LIN {X 0,Y 676.255,Z 793.272,A -85,B 0,C 180,E1 -4017.987,E2 -4017.987} C_VEL
LIN {X 0,Y 675.529,Z 814.442,A -85,B 0,C 180,E1 -4018.503,E2 -4018.503} C_VEL
LIN {X 0,Y 674.622,Z 838.545,A -85,B 0,C 180,E1 -4019.247,E2 -4019.247} C_VEL
LIN {X 0,Y 673.655,Z 859.341,A -85,B 0,C 180,E1 -4020.036,E2 -4020.036} C_VEL
LIN {X 0,Y 672.656,Z 880.169,A -85,B 0,C 180,E1 -4020.961,E2 -4020.961} C_VEL
LIN {X 0,Y 671.429,Z 902.312,A -85,B 0,C 180,E1 -4022.121,E2 -4022.121} C_VEL
LIN {X 0,Y 670.354,Z 922.188,A -85,B 0,C 180,E1 -4023.323,E2 -4023.323} C_VEL
LIN {X 0,Y 669.168,Z 942.613,A -85,B 0,C 180,E1 -4024.748,E2 -4024.748} C_VEL
LIN {X 0,Y 668.228,Z 959.686,A -85,B 0,C 180,E1 -4026.101,E2 -4026.101} C_VEL
LIN {X 0,Y 667.192,Z 978.605,A -85,B 0,C 180,E1 -4027.811,E2 -4027.811} C_VEL
LIN {X 0,Y 666.434,Z 993.632,A -85,B 0,C 180,E1 -4029.354,E2 -4029.354} C_VEL
LIN {X 0,Y 665.654,Z 1009.818,A -85,B 0,C 180,E1 -4031.249,E2 -4031.249} C_VEL
LIN {X 0,Y 665.144,Z 1022.543,A -85,B 0,C 180,E1 -4032.957,E2 -4032.957} C_VEL
LIN {X 0,Y 664.665,Z 1035.765,A -85,B 0,C 180,E1 -4035.004,E2 -4035.004} C_VEL
LIN {X 0,Y 664.369,Z 1045.92,A -85,B 0,C 180,E1 -4036.844,E2 -4036.844} C_VEL
LIN {X 0,Y 664.132,Z 1055.929,A -85,B 0,C 180,E1 -4039.001,E2 -4039.001} C_VEL
LIN {X 0,Y 664.022,Z 1062.817,A -85,B 0,C 180,E1 -4040.815,E2 -4040.815} C_VEL
LIN {X 0,Y 663.962,Z 1069.244,A -85,B 0,C 180,E1 -4042.907,E2 -4042.907} C_VEL
LIN {X 0,Y 663.925,Z 1073.656,A -85,B 0,C 180,E1 -4044.902,E2 -4044.902} C_VEL
LIN {X 0,Y 663.917,Z 1076.574,A -85,B 0,C 180,E1 -4046.806,E2 -4046.806} C_VEL
LIN {X 0,Y 663.91,Z 1078.26,A -85,B 0,C 180,E1 -4049.051,E2 -4049.051} C_VEL
LIN {X 0,Y 663.905,Z 1078.283,A -85,B 0,C 180,E1 -4050.863,E2 -4050.863} C_VEL
LIN {X 0,Y 663.916,Z 1076.799,A -85,B 0,C 180,E1 -4053.021,E2 -4053.021} C_VEL
LIN {X 0,Y 663.925,Z 1073.815,A -85,B 0,C 180,E1 -4055.011,E2 -4055.011} C_VEL
LIN {X 0,Y 663.956,Z 1069.451,A -85,B 0,C 180,E1 -4057.006,E2 -4057.006} C_VEL
LIN {X 0,Y 664.011,Z 1063.12,A -85,B 0,C 180,E1 -4059.097,E2 -4059.097} C_VEL
LIN {X 0,Y 664.128,Z 1056.187,A -85,B 0,C 180,E1 -4060.935,E2 -4060.935} C_VEL
LIN {X 0,Y 664.355,Z 1046.484,A -85,B 0,C 180,E1 -4063.047,E2 -4063.047} C_VEL
LIN {X 0,Y 664.649,Z 1036.288,A -85,B 0,C 180,E1 -4064.907,E2 -4064.907} C_VEL
LIN {X 0,Y 665.121,Z 1023.161,A -85,B 0,C 180,E1 -4066.956,E2 -4066.956} C_VEL
LIN {X 0,Y 665.624,Z 1010.525,A -85,B 0,C 180,E1 -4068.661,E2 -4068.661} C_VEL
LIN {X 0,Y 666.403,Z 994.378,A -85,B 0,C 180,E1 -4070.565,E2 -4070.565} C_VEL
LIN {X 0,Y 667.168,Z 979.013,A -85,B 0,C 180,E1 -4072.149,E2 -4072.149} C_VEL
LIN {X 0,Y 668.189,Z 960.507,A -85,B 0,C 180,E1 -4073.83,E2 -4073.83} C_VEL
LIN {X 0,Y 669.128,Z 943.221,A -85,B 0,C 180,E1 -4075.206,E2 -4075.206} C_VEL
LIN {X 0,Y 670.317,Z 922.91,A -85,B 0,C 180,E1 -4076.631,E2 -4076.631} C_VEL
LIN {X 0,Y 671.389,Z 903.049,A -85,B 0,C 180,E1 -4077.837,E2 -4077.837} C_VEL
LIN {X 0,Y 672.604,Z 881.269,A -85,B 0,C 180,E1 -4078.988,E2 -4078.988} C_VEL
LIN {X 0,Y 673.605,Z 860.478,A -85,B 0,C 180,E1 -4079.917,E2 -4079.917} C_VEL
LIN {X 0,Y 674.538,Z 840.352,A -85,B 0,C 180,E1 -4080.688,E2 -4080.688} C_VEL
LIN {X 0,Y 675.503,Z 815.102,A -85,B 0,C 180,E1 -4081.479,E2 -4081.479} C_VEL
LIN {X 0,Y 676.234,Z 793.804,A -85,B 0,C 180,E1 -4082.002,E2 -4082.002} C_VEL
LIN {X 0,Y 676.909,Z 768.362,A -85,B 0,C 180,E1 -4082.466,E2 -4082.466} C_VEL
LIN {X 0,Y 677.775,Z 687.285,A -85,B 0,C 180,E1 -4083.452,E2 -4083.452} C_VEL
LIN {X 0,Y 680.315,Z 434.11,A -85,B 0,C 180,E1 -4086.498,E2 -4086.498} C_VEL
LIN {X 0,Y 680.519,Z 397.747,A -85,B 0,C 180,E1 -4086.954,E2 -4086.954} C_VEL
LIN {X 0,Y 675.309,Z 375.993,A -85,B 0,C 180,E1 -4087.591,E2 -4087.591} C_VEL
LIN {X 0,Y 675.512,Z 367.277,A -85,B 0,C 180,E1 -4088.256,E2 -4088.256} C_VEL
LIN {X 0,Y 667.876,Z 347.353,A -85,B 0,C 180,E1 -4090.356,E2 -4090.356} C_VEL
LIN {X 0,Y 664.606,Z 338.448,A -85,B 0,C 180,E1 -4091.345,E2 -4091.345} C_VEL
LIN {X 0,Y 664.58,Z 338.444,A -85,B 0,C 180,E1 -4094.035,E2 -4094.035} C_VEL
LIN {X 0,Y 664.647,Z 338.444,A -85,B 0,C 180,E1 -4097.04,E2 -4097.04} C_VEL
LIN {X 0,Y 664.579,Z 338.44,A -85,B 0,C 180,E1 -4099.913,E2 -4099.913} C_VEL
LIN {X 0,Y 664.625,Z 338.437,A -85,B 0,C 180,E1 -4102.735,E2 -4102.735} C_VEL
LIN {X 0,Y 664.588,Z 338.439,A -85,B 0,C 180,E1 -4105.842,E2 -4105.842} C_VEL
LIN {X 0,Y 664.593,Z 338.436,A -85,B 0,C 180,E1 -4108.546,E2 -4108.546} C_VEL
LIN {X 0,Y 664.605,Z 338.436,A -85,B 0,C 180,E1 -4111.711,E2 -4111.711} C_VEL
LIN {X 0,Y 664.584,Z 338.441,A -85,B 0,C 180,E1 -4114.418,E2 -4114.418} C_VEL
LIN {X 0,Y 664.651,Z 338.44,A -85,B 0,C 180,E1 -4117.472,E2 -4117.472} C_VEL
LIN {X 0,Y 664.579,Z 338.438,A -85,B 0,C 180,E1 -4120.396,E2 -4120.396} C_VEL
LIN {X 0,Y 664.647,Z 338.438,A -85,B 0,C 180,E1 -4123.301,E2 -4123.301} C_VEL
LIN {X 0,Y 664.586,Z 338.442,A -85,B 0,C 180,E1 -4126.248,E2 -4126.248} C_VEL
LIN {X 0,Y 664.604,Z 338.433,A -85,B 0,C 180,E1 -4128.985,E2 -4128.985} C_VEL
LIN {X 0,Y 664.6,Z 338.434,A -85,B 0,C 180,E1 -4132.131,E2 -4132.131} C_VEL
LIN {X 0,Y 664.589,Z 338.44,A -85,B 0,C 180,E1 -4134.869,E2 -4134.869} C_VEL
LIN {X 0,Y 664.636,Z 338.436,A -85,B 0,C 180,E1 -4137.931,E2 -4137.931} C_VEL
LIN {X 0,Y 664.582,Z 338.439,A -85,B 0,C 180,E1 -4140.776,E2 -4140.776} C_VEL
LIN {X 0,Y 664.649,Z 338.435,A -85,B 0,C 180,E1 -4143.709,E2 -4143.709} C_VEL
LIN {X 0,Y 664.584,Z 338.434,A -85,B 0,C 180,E1 -4146.653,E2 -4146.653} C_VEL
LIN {X 0,Y 664.618,Z 338.439,A -85,B 0,C 180,E1 -4149.438,E2 -4149.438} C_VEL
LIN {X 0,Y 664.594,Z 338.443,A -85,B 0,C 180,E1 -4152.601,E2 -4152.601} C_VEL
LIN {X 0,Y 664.598,Z 338.435,A -85,B 0,C 180,E1 -4155.355,E2 -4155.355} C_VEL
LIN {X 0,Y 664.611,Z 338.441,A -85,B 0,C 180,E1 -4158.509,E2 -4158.509} C_VEL
LIN {X 0,Y 664.589,Z 338.439,A -85,B 0,C 180,E1 -4161.259,E2 -4161.259} C_VEL
LIN {X 0,Y 664.647,Z 338.435,A -85,B 0,C 180,E1 -4164.264,E2 -4164.264} C_VEL
LIN {X 0,Y 664.585,Z 338.438,A -85,B 0,C 180,E1 -4167.121,E2 -4167.121} C_VEL
LIN {X 0,Y 664.643,Z 338.438,A -85,B 0,C 180,E1 -4169.965,E2 -4169.965} C_VEL
LIN {X 0,Y 664.591,Z 338.442,A -85,B 0,C 180,E1 -4173.069,E2 -4173.069} C_VEL
LIN {X 0,Y 664.624,Z 338.437,A -85,B 0,C 180,E1 -4175.926,E2 -4175.926} C_VEL
LIN {X 0,Y 664.65,Z 338.441,A -85,B 0,C 180,E1 -4176.376,E2 -4176.376} C_VEL
LIN {X 0,Y 663.65,Z 338.574,A -85,B 0,C 180,E1 -4177.041,E2 -4177.041} C_VEL
LIN {X 0,Y 657.182,Z 339.37,A -85,B 0,C 180,E1 -4178.902,E2 -4178.902} C_VEL
LIN {X 0,Y 656.649,Z 339.431,A -85,B 0,C 180,E1 -4179.386,E2 -4179.386} C_VEL
LIN {X 0,Y 656.711,Z 339.43,A -85,B 0,C 180,E1 -4182.298,E2 -4182.298} C_VEL
LIN {X 0,Y 656.652,Z 339.432,A -85,B 0,C 180,E1 -4185.325,E2 -4185.325} C_VEL
LIN {X 0,Y 656.7,Z 339.431,A -85,B 0,C 180,E1 -4188.252,E2 -4188.252} C_VEL
LIN {X 0,Y 656.721,Z 339.5,A -85,B 0,C 180,E1 -4190.391,E2 -4190.391} C_VEL
LIN {X 0,Y 660.252,Z 349.072,A -85,B 0,C 180,E1 -4191.479,E2 -4191.479} C_VEL
LIN {X 0,Y 674.214,Z 372.691,A -85,B 0,C 180,E1 -4192.737,E2 -4192.737} C_VEL
LIN {X 0,Y 672.117,Z 564.734,A -85,B 0,C 180,E1 -4195.097,E2 -4195.097} C_VEL
LIN {X 0,Y 670.164,Z 737.365,A -85,B 0,C 180,E1 -4197.196,E2 -4197.196} C_VEL
LIN {X 0,Y 669.465,Z 762.862,A -85,B 0,C 180,E1 -4197.658,E2 -4197.658} C_VEL
LIN {X 0,Y 668.692,Z 783.876,A -85,B 0,C 180,E1 -4198.172,E2 -4198.172} C_VEL
LIN {X 0,Y 667.724,Z 807.392,A -85,B 0,C 180,E1 -4198.894,E2 -4198.894} C_VEL
LIN {X 0,Y 666.664,Z 828.321,A -85,B 0,C 180,E1 -4199.689,E2 -4199.689} C_VEL
LIN {X 0,Y 665.591,Z 849.051,A -85,B 0,C 180,E1 -4200.612,E2 -4200.612} C_VEL
LIN {X 0,Y 664.244,Z 871.561,A -85,B 0,C 180,E1 -4201.793,E2 -4201.793} C_VEL
LIN {X 0,Y 663.077,Z 891.047,A -85,B 0,C 180,E1 -4202.976,E2 -4202.976} C_VEL
LIN {X 0,Y 661.793,Z 911.734,A -85,B 0,C 180,E1 -4204.422,E2 -4204.422} C_VEL
LIN {X 0,Y 660.725,Z 928.876,A -85,B 0,C 180,E1 -4205.788,E2 -4205.788} C_VEL
LIN {X 0,Y 659.58,Z 948.163,A -85,B 0,C 180,E1 -4207.541,E2 -4207.541} C_VEL
LIN {X 0,Y 658.72,Z 963.223,A -85,B 0,C 180,E1 -4209.102,E2 -4209.102} C_VEL
LIN {X 0,Y 657.874,Z 979.475,A -85,B 0,C 180,E1 -4211.019,E2 -4211.019} C_VEL
LIN {X 0,Y 657.298,Z 992.211,A -85,B 0,C 180,E1 -4212.744,E2 -4212.744} C_VEL
LIN {X 0,Y 656.756,Z 1005.695,A -85,B 0,C 180,E1 -4214.851,E2 -4214.851} C_VEL
LIN {X 0,Y 656.432,Z 1015.336,A -85,B 0,C 180,E1 -4216.613,E2 -4216.613} C_VEL
LIN {X 0,Y 656.186,Z 1024.942,A -85,B 0,C 180,E1 -4218.664,E2 -4218.664} C_VEL
LIN {X 0,Y 656.047,Z 1032.359,A -85,B 0,C 180,E1 -4220.614,E2 -4220.614} C_VEL
LIN {X 0,Y 655.948,Z 1038.123,A -85,B 0,C 180,E1 -4222.467,E2 -4222.467} C_VEL
LIN {X 0,Y 655.915,Z 1043.254,A -85,B 0,C 180,E1 -4224.664,E2 -4224.664} C_VEL
LIN {X 0,Y 655.912,Z 1046.179,A -85,B 0,C 180,E1 -4226.504,E2 -4226.504} C_VEL
LIN {X 0,Y 655.898,Z 1048.129,A -85,B 0,C 180,E1 -4228.602,E2 -4228.602} C_VEL
LIN {X 0,Y 655.894,Z 1048.362,A -85,B 0,C 180,E1 -4230.612,E2 -4230.612} C_VEL
LIN {X 0,Y 655.907,Z 1047.397,A -85,B 0,C 180,E1 -4232.446,E2 -4232.446} C_VEL
LIN {X 0,Y 655.918,Z 1044.691,A -85,B 0,C 180,E1 -4234.634,E2 -4234.634} C_VEL
LIN {X 0,Y 655.93,Z 1040.795,A -85,B 0,C 180,E1 -4236.565,E2 -4236.565} C_VEL
LIN {X 0,Y 655.988,Z 1035.585,A -85,B 0,C 180,E1 -4238.503,E2 -4238.503} C_VEL
LIN {X 0,Y 656.123,Z 1028.137,A -85,B 0,C 180,E1 -4240.626,E2 -4240.626} C_VEL
LIN {X 0,Y 656.298,Z 1020.469,A -85,B 0,C 180,E1 -4242.422,E2 -4242.422} C_VEL
LIN {X 0,Y 656.627,Z 1009.634,A -85,B 0,C 180,E1 -4244.552,E2 -4244.552} C_VEL
LIN {X 0,Y 657.016,Z 998.83,A -85,B 0,C 180,E1 -4246.353,E2 -4246.353} C_VEL
LIN {X 0,Y 657.631,Z 985.069,A -85,B 0,C 180,E1 -4248.345,E2 -4248.345} C_VEL
LIN {X 0,Y 658.286,Z 971.227,A -85,B 0,C 180,E1 -4250.077,E2 -4250.077} C_VEL
LIN {X 0,Y 659.186,Z 955.439,A -85,B 0,C 180,E1 -4251.825,E2 -4251.825} C_VEL
LIN {X 0,Y 660.116,Z 938.8,A -85,B 0,C 180,E1 -4253.429,E2 -4253.429} C_VEL
LIN {X 0,Y 661.281,Z 920.46,A -85,B 0,C 180,E1 -4255,E2 -4255} C_VEL
LIN {X 0,Y 662.437,Z 901.028,A -85,B 0,C 180,E1 -4256.441,E2 -4256.441} C_VEL
LIN {X 0,Y 663.767,Z 880.336,A -85,B 0,C 180,E1 -4257.79,E2 -4257.79} C_VEL
LIN {X 0,Y 664.964,Z 859.37,A -85,B 0,C 180,E1 -4258.959,E2 -4258.959} C_VEL
LIN {X 0,Y 666.25,Z 837.109,A -85,B 0,C 180,E1 -4260.034,E2 -4260.034} C_VEL
LIN {X 0,Y 667.326,Z 815.541,A -85,B 0,C 180,E1 -4260.899,E2 -4260.899} C_VEL
LIN {X 0,Y 668.244,Z 795.426,A -85,B 0,C 180,E1 -4261.581,E2 -4261.581} C_VEL
LIN {X 0,Y 669.182,Z 770.572,A -85,B 0,C 180,E1 -4262.26,E2 -4262.26} C_VEL
LIN {X 0,Y 669.871,Z 748.473,A -85,B 0,C 180,E1 -4262.713,E2 -4262.713} C_VEL
LIN {X 0,Y 670.423,Z 721.817,A -85,B 0,C 180,E1 -4263.101,E2 -4263.101} C_VEL
LIN {X 0,Y 673.237,Z 466.687,A -85,B 0,C 180,E1 -4266.188,E2 -4266.188} C_VEL
LIN {X 0,Y 674.129,Z 372.539,A -85,B 0,C 180,E1 -4267.361,E2 -4267.361} C_VEL
LIN {X 0,Y 662.253,Z 352.49,A -85,B 0,C 180,E1 -4268.425,E2 -4268.425} C_VEL
LIN {X 0,Y 659.963,Z 348.582,A -85,B 0,C 180,E1 -4268.646,E2 -4268.646} C_VEL
LIN {X 0,Y 656.696,Z 339.429,A -85,B 0,C 180,E1 -4269.743,E2 -4269.743} C_VEL
LIN {X 0,Y 656.642,Z 339.436,A -85,B 0,C 180,E1 -4272.539,E2 -4272.539} C_VEL
LIN {X 0,Y 656.706,Z 339.422,A -85,B 0,C 180,E1 -4275.444,E2 -4275.444} C_VEL
LIN {X 0,Y 656.644,Z 339.408,A -85,B 0,C 180,E1 -4278.401,E2 -4278.401} C_VEL
LIN {X 0,Y 656.666,Z 339.432,A -85,B 0,C 180,E1 -4281.145,E2 -4281.145} C_VEL
LIN {X 0,Y 656.657,Z 339.431,A -85,B 0,C 180,E1 -4284.324,E2 -4284.324} C_VEL
LIN {X 0,Y 656.651,Z 339.432,A -85,B 0,C 180,E1 -4287.07,E2 -4287.07} C_VEL
LIN {X 0,Y 656.679,Z 339.429,A -85,B 0,C 180,E1 -4290.217,E2 -4290.217} C_VEL
LIN {X 0,Y 656.643,Z 339.424,A -85,B 0,C 180,E1 -4293.014,E2 -4293.014} C_VEL
LIN {X 0,Y 656.709,Z 339.42,A -85,B 0,C 180,E1 -4296.013,E2 -4296.013} C_VEL
LIN {X 0,Y 656.639,Z 339.431,A -85,B 0,C 180,E1 -4298.939,E2 -4298.939} C_VEL
LIN {X 0,Y 656.702,Z 339.43,A -85,B 0,C 180,E1 -4301.823,E2 -4301.823} C_VEL
LIN {X 0,Y 656.643,Z 339.422,A -85,B 0,C 180,E1 -4304.887,E2 -4304.887} C_VEL
LIN {X 0,Y 656.665,Z 339.434,A -85,B 0,C 180,E1 -4307.602,E2 -4307.602} C_VEL
LIN {X 0,Y 656.654,Z 339.429,A -85,B 0,C 180,E1 -4310.8,E2 -4310.8} C_VEL
LIN {X 0,Y 656.649,Z 339.427,A -85,B 0,C 180,E1 -4313.53,E2 -4313.53} C_VEL
LIN {X 0,Y 656.675,Z 339.426,A -85,B 0,C 180,E1 -4316.683,E2 -4316.683} C_VEL
LIN {X 0,Y 656.641,Z 339.426,A -85,B 0,C 180,E1 -4319.477,E2 -4319.477} C_VEL
LIN {X 0,Y 656.708,Z 339.418,A -85,B 0,C 180,E1 -4322.443,E2 -4322.443} C_VEL
LIN {X 0,Y 656.639,Z 339.431,A -85,B 0,C 180,E1 -4325.417,E2 -4325.417} C_VEL
LIN {X 0,Y 656.709,Z 339.422,A -85,B 0,C 180,E1 -4328.317,E2 -4328.317} C_VEL
LIN {X 0,Y 656.642,Z 339.427,A -85,B 0,C 180,E1 -4331.328,E2 -4331.328} C_VEL
LIN {X 0,Y 656.67,Z 339.431,A -85,B 0,C 180,E1 -4334.101,E2 -4334.101} C_VEL
LIN {X 0,Y 656.65,Z 339.425,A -85,B 0,C 180,E1 -4337.273,E2 -4337.273} C_VEL
LIN {X 0,Y 656.648,Z 339.431,A -85,B 0,C 180,E1 -4339.943,E2 -4339.943} C_VEL
LIN {X 0,Y 656.685,Z 339.426,A -85,B 0,C 180,E1 -4343.037,E2 -4343.037} C_VEL
LIN {X 0,Y 656.64,Z 339.43,A -85,B 0,C 180,E1 -4345.85,E2 -4345.85} C_VEL
LIN {X 0,Y 656.717,Z 339.428,A -85,B 0,C 180,E1 -4348.859,E2 -4348.859} C_VEL
LIN {X 0,Y 656.638,Z 339.428,A -85,B 0,C 180,E1 -4351.794,E2 -4351.794} C_VEL
LIN {X 0,Y 656.689,Z 339.428,A -85,B 0,C 180,E1 -4354.607,E2 -4354.607} C_VEL
LIN {X 0,Y 656.649,Z 339.431,A -85,B 0,C 180,E1 -4357.645,E2 -4357.645} C_VEL
LIN {X 0,Y 656.648,Z 339.416,A -85,B 0,C 180,E1 -4360.328,E2 -4360.328} C_VEL
LIN {X 0,Y 656.671,Z 339.428,A -85,B 0,C 180,E1 -4363.492,E2 -4363.492} C_VEL
LIN {X 0,Y 656.642,Z 339.431,A -85,B 0,C 180,E1 -4366.265,E2 -4366.265} C_VEL
LIN {X 0,Y 656.658,Z 339.573,A -85,B 0,C 180,E1 -4368.184,E2 -4368.184} C_VEL
LIN {X 0,Y 666.139,Z 364.38,A -85,B 0,C 180,E1 -4370.899,E2 -4370.899} C_VEL
LIN {X 0,Y 668.561,Z 371.173,A -85,B 0,C 180,E1 -4371.6,E2 -4371.6} C_VEL
LIN {X 0,Y 668.498,Z 376.61,A -85,B 0,C 180,E1 -4371.992,E2 -4371.992} C_VEL
LIN {X 0,Y 674.27,Z 401.056,A -85,B 0,C 180,E1 -4372.692,E2 -4372.692} C_VEL
LIN {X 0,Y 671.314,Z 665.846,A -85,B 0,C 180,E1 -4375.914,E2 -4375.914} C_VEL
LIN {X 0,Y 670.159,Z 767.706,A -85,B 0,C 180,E1 -4377.156,E2 -4377.156} C_VEL
LIN {X 0,Y 669.461,Z 793.009,A -85,B 0,C 180,E1 -4377.616,E2 -4377.616} C_VEL
LIN {X 0,Y 668.687,Z 814.006,A -85,B 0,C 180,E1 -4378.131,E2 -4378.131} C_VEL
LIN {X 0,Y 667.733,Z 837.257,A -85,B 0,C 180,E1 -4378.844,E2 -4378.844} C_VEL
LIN {X 0,Y 666.671,Z 858.206,A -85,B 0,C 180,E1 -4379.639,E2 -4379.639} C_VEL
LIN {X 0,Y 665.63,Z 878.269,A -85,B 0,C 180,E1 -4380.53,E2 -4380.53} C_VEL
LIN {X 0,Y 664.255,Z 901.416,A -85,B 0,C 180,E1 -4381.739,E2 -4381.739} C_VEL
LIN {X 0,Y 663.095,Z 920.727,A -85,B 0,C 180,E1 -4382.91,E2 -4382.91} C_VEL
LIN {X 0,Y 661.775,Z 942.002,A -85,B 0,C 180,E1 -4384.398,E2 -4384.398} C_VEL
LIN {X 0,Y 660.695,Z 959.399,A -85,B 0,C 180,E1 -4385.787,E2 -4385.787} C_VEL
LIN {X 0,Y 659.552,Z 978.604,A -85,B 0,C 180,E1 -4387.54,E2 -4387.54} C_VEL
LIN {X 0,Y 658.705,Z 993.63,A -85,B 0,C 180,E1 -4389.101,E2 -4389.101} C_VEL
LIN {X 0,Y 657.857,Z 1009.82,A -85,B 0,C 180,E1 -4391.018,E2 -4391.018} C_VEL
LIN {X 0,Y 657.284,Z 1022.521,A -85,B 0,C 180,E1 -4392.744,E2 -4392.744} C_VEL
LIN {X 0,Y 656.744,Z 1035.973,A -85,B 0,C 180,E1 -4394.855,E2 -4394.855} C_VEL
LIN {X 0,Y 656.42,Z 1046.022,A -85,B 0,C 180,E1 -4396.702,E2 -4396.702} C_VEL
LIN {X 0,Y 656.155,Z 1056.164,A -85,B 0,C 180,E1 -4398.924,E2 -4398.924} C_VEL
LIN {X 0,Y 656.032,Z 1063.12,A -85,B 0,C 180,E1 -4400.791,E2 -4400.791} C_VEL
LIN {X 0,Y 655.964,Z 1069.45,A -85,B 0,C 180,E1 -4402.908,E2 -4402.908} C_VEL
LIN {X 0,Y 655.926,Z 1073.815,A -85,B 0,C 180,E1 -4404.928,E2 -4404.928} C_VEL
LIN {X 0,Y 655.917,Z 1076.799,A -85,B 0,C 180,E1 -4406.941,E2 -4406.941} C_VEL
LIN {X 0,Y 655.906,Z 1078.283,A -85,B 0,C 180,E1 -4409.126,E2 -4409.126} C_VEL
LIN {X 0,Y 655.91,Z 1078.26,A -85,B 0,C 180,E1 -4410.961,E2 -4410.961} C_VEL
LIN {X 0,Y 655.918,Z 1076.687,A -85,B 0,C 180,E1 -4413.146,E2 -4413.146} C_VEL
LIN {X 0,Y 655.925,Z 1073.815,A -85,B 0,C 180,E1 -4415.072,E2 -4415.072} C_VEL
LIN {X 0,Y 655.964,Z 1069.428,A -85,B 0,C 180,E1 -4417.102,E2 -4417.102} C_VEL
LIN {X 0,Y 656.032,Z 1063.119,A -85,B 0,C 180,E1 -4419.209,E2 -4419.209} C_VEL
LIN {X 0,Y 656.155,Z 1056.163,A -85,B 0,C 180,E1 -4421.076,E2 -4421.076} C_VEL
LIN {X 0,Y 656.42,Z 1046.025,A -85,B 0,C 180,E1 -4423.298,E2 -4423.298} C_VEL
LIN {X 0,Y 656.745,Z 1035.974,A -85,B 0,C 180,E1 -4425.145,E2 -4425.145} C_VEL
LIN {X 0,Y 657.284,Z 1022.524,A -85,B 0,C 180,E1 -4427.256,E2 -4427.256} C_VEL
LIN {X 0,Y 657.857,Z 1009.82,A -85,B 0,C 180,E1 -4428.981,E2 -4428.981} C_VEL
LIN {X 0,Y 658.706,Z 993.631,A -85,B 0,C 180,E1 -4430.899,E2 -4430.899} C_VEL
LIN {X 0,Y 659.552,Z 978.606,A -85,B 0,C 180,E1 -4432.46,E2 -4432.46} C_VEL
LIN {X 0,Y 660.724,Z 958.846,A -85,B 0,C 180,E1 -4434.259,E2 -4434.259} C_VEL
LIN {X 0,Y 661.83,Z 941.236,A -85,B 0,C 180,E1 -4435.66,E2 -4435.66} C_VEL
LIN {X 0,Y 663.13,Z 919.986,A -85,B 0,C 180,E1 -4437.137,E2 -4437.137} C_VEL
LIN {X 0,Y 664.304,Z 900.684,A -85,B 0,C 180,E1 -4438.303,E2 -4438.303} C_VEL
LIN {X 0,Y 665.679,Z 877.271,A -85,B 0,C 180,E1 -4439.517,E2 -4439.517} C_VEL
LIN {X 0,Y 666.707,Z 857.463,A -85,B 0,C 180,E1 -4440.392,E2 -4440.392} C_VEL
LIN {X 0,Y 667.886,Z 833.799,A -85,B 0,C 180,E1 -4441.271,E2 -4441.271} C_VEL
LIN {X 0,Y 668.755,Z 812.388,A -85,B 0,C 180,E1 -4441.913,E2 -4441.913} C_VEL
LIN {X 0,Y 669.581,Z 790.08,A -85,B 0,C 180,E1 -4442.449,E2 -4442.449} C_VEL
LIN {X 0,Y 670.189,Z 765.257,A -85,B 0,C 180,E1 -4442.878,E2 -4442.878} C_VEL
LIN {X 0,Y 672.805,Z 526.422,A -85,B 0,C 180,E1 -4445.774,E2 -4445.774} C_VEL
LIN {X 0,Y 674.093,Z 399.553,A -85,B 0,C 180,E1 -4447.339,E2 -4447.339} C_VEL
LIN {X 0,Y 668.4,Z 375.759,A -85,B 0,C 180,E1 -4448.048,E2 -4448.048} C_VEL
LIN {X 0,Y 668.439,Z 370.569,A -85,B 0,C 180,E1 -4448.456,E2 -4448.456} C_VEL
LIN {X 0,Y 660.223,Z 348.835,A -85,B 0,C 180,E1 -4450.778,E2 -4450.778} C_VEL
LIN {X 0,Y 656.641,Z 339.434,A -85,B 0,C 180,E1 -4451.833,E2 -4451.833} C_VEL
LIN {X 0,Y 656.699,Z 339.43,A -85,B 0,C 180,E1 -4454.704,E2 -4454.704} C_VEL
LIN {X 0,Y 656.646,Z 339.43,A -85,B 0,C 180,E1 -4457.735,E2 -4457.735} C_VEL
LIN {X 0,Y 656.66,Z 339.426,A -85,B 0,C 180,E1 -4460.47,E2 -4460.47} C_VEL
LIN {X 0,Y 656.654,Z 339.403,A -85,B 0,C 180,E1 -4463.677,E2 -4463.677} C_VEL
LIN {X 0,Y 656.651,Z 339.425,A -85,B 0,C 180,E1 -4466.444,E2 -4466.444} C_VEL
LIN {X 0,Y 656.684,Z 339.428,A -85,B 0,C 180,E1 -4469.533,E2 -4469.533} C_VEL
LIN {X 0,Y 656.642,Z 339.422,A -85,B 0,C 180,E1 -4472.326,E2 -4472.326} C_VEL
LIN {X 0,Y 656.712,Z 339.425,A -85,B 0,C 180,E1 -4475.343,E2 -4475.343} C_VEL
LIN {X 0,Y 656.643,Z 339.431,A -85,B 0,C 180,E1 -4478.283,E2 -4478.283} C_VEL
LIN {X 0,Y 656.701,Z 339.424,A -85,B 0,C 180,E1 -4481.168,E2 -4481.168} C_VEL
LIN {X 0,Y 656.645,Z 339.427,A -85,B 0,C 180,E1 -4484.23,E2 -4484.23} C_VEL
LIN {X 0,Y 656.674,Z 339.428,A -85,B 0,C 180,E1 -4487.033,E2 -4487.033} C_VEL
LIN {X 0,Y 656.654,Z 339.433,A -85,B 0,C 180,E1 -4490.181,E2 -4490.181} C_VEL
LIN {X 0,Y 656.652,Z 339.418,A -85,B 0,C 180,E1 -4492.915,E2 -4492.915} C_VEL
LIN {X 0,Y 656.675,Z 339.427,A -85,B 0,C 180,E1 -4496.071,E2 -4496.071} C_VEL
LIN {X 0,Y 656.646,Z 339.428,A -85,B 0,C 180,E1 -4498.866,E2 -4498.866} C_VEL
LIN {X 0,Y 656.709,Z 339.422,A -85,B 0,C 180,E1 -4501.832,E2 -4501.832} C_VEL
LIN {X 0,Y 656.643,Z 339.43,A -85,B 0,C 180,E1 -4504.804,E2 -4504.804} C_VEL
LIN {X 0,Y 656.711,Z 339.419,A -85,B 0,C 180,E1 -4507.788,E2 -4507.788} C_VEL
LIN {X 0,Y 656.645,Z 339.423,A -85,B 0,C 180,E1 -4510.795,E2 -4510.795} C_VEL
LIN {X 0,Y 656.704,Z 339.427,A -85,B 0,C 180,E1 -4513.734,E2 -4513.734} C_VEL
LIN {X 0,Y 656.653,Z 339.431,A -85,B 0,C 180,E1 -4516.726,E2 -4516.726} C_VEL
LIN {X 0,Y 656.67,Z 339.425,A -85,B 0,C 180,E1 -4519.519,E2 -4519.519} C_VEL
LIN {X 0,Y 656.665,Z 339.43,A -85,B 0,C 180,E1 -4522.67,E2 -4522.67} C_VEL
LIN {X 0,Y 656.656,Z 339.428,A -85,B 0,C 180,E1 -4525.45,E2 -4525.45} C_VEL
LIN {X 0,Y 656.687,Z 339.429,A -85,B 0,C 180,E1 -4528.562,E2 -4528.562} C_VEL
LIN {X 0,Y 656.648,Z 339.422,A -85,B 0,C 180,E1 -4531.384,E2 -4531.384} C_VEL
LIN {X 0,Y 656.709,Z 339.424,A -85,B 0,C 180,E1 -4534.394,E2 -4534.394} C_VEL
LIN {X 0,Y 656.647,Z 339.424,A -85,B 0,C 180,E1 -4537.358,E2 -4537.358} C_VEL
LIN {X 0,Y 656.649,Z 339.431,A -85,B 0,C 180,E1 -4539.386,E2 -4539.386} C_VEL
LIN {X 0,Y 655.676,Z 339.554,A -85,B 0,C 180,E1 -4540.058,E2 -4540.058} C_VEL
LIN {X 0,Y 649.313,Z 340.353,A -85,B 0,C 180,E1 -4541.942,E2 -4541.942} C_VEL
LIN {X 0,Y 648.772,Z 340.416,A -85,B 0,C 180,E1 -4542.432,E2 -4542.432} C_VEL
LIN {X 0,Y 648.71,Z 340.421,A -85,B 0,C 180,E1 -4545.407,E2 -4545.407} C_VEL
LIN {X 0,Y 648.773,Z 340.421,A -85,B 0,C 180,E1 -4548.375,E2 -4548.375} C_VEL
LIN {X 0,Y 648.738,Z 340.547,A -85,B 0,C 180,E1 -4549.877,E2 -4549.877} C_VEL
LIN {X 0,Y 652.07,Z 349.421,A -85,B 0,C 180,E1 -4550.905,E2 -4550.905} C_VEL
LIN {X 0,Y 664.266,Z 369.643,A -85,B 0,C 180,E1 -4552.035,E2 -4552.035} C_VEL
LIN {X 0,Y 667.911,Z 376.42,A -85,B 0,C 180,E1 -4552.371,E2 -4552.371} C_VEL
LIN {X 0,Y 664.936,Z 618.068,A -85,B 0,C 180,E1 -4555.351,E2 -4555.351} C_VEL
LIN {X 0,Y 663.446,Z 737.809,A -85,B 0,C 180,E1 -4556.825,E2 -4556.825} C_VEL
LIN {X 0,Y 662.694,Z 763.145,A -85,B 0,C 180,E1 -4557.29,E2 -4557.29} C_VEL
LIN {X 0,Y 661.868,Z 783.849,A -85,B 0,C 180,E1 -4557.802,E2 -4557.802} C_VEL
LIN {X 0,Y 660.804,Z 807.405,A -85,B 0,C 180,E1 -4558.531,E2 -4558.531} C_VEL
LIN {X 0,Y 659.597,Z 829.462,A -85,B 0,C 180,E1 -4559.38,E2 -4559.38} C_VEL
LIN {X 0,Y 658.373,Z 851.379,A -85,B 0,C 180,E1 -4560.373,E2 -4560.373} C_VEL
LIN {X 0,Y 656.929,Z 873.189,A -85,B 0,C 180,E1 -4561.549,E2 -4561.549} C_VEL
LIN {X 0,Y 655.612,Z 893.704,A -85,B 0,C 180,E1 -4562.821,E2 -4562.821} C_VEL
LIN {X 0,Y 654.217,Z 913.869,A -85,B 0,C 180,E1 -4564.275,E2 -4564.275} C_VEL
LIN {X 0,Y 652.984,Z 932.753,A -85,B 0,C 180,E1 -4565.82,E2 -4565.82} C_VEL
LIN {X 0,Y 651.831,Z 950.018,A -85,B 0,C 180,E1 -4567.45,E2 -4567.45} C_VEL
LIN {X 0,Y 650.841,Z 966.6,A -85,B 0,C 180,E1 -4569.214,E2 -4569.214} C_VEL
LIN {X 0,Y 649.962,Z 981.585,A -85,B 0,C 180,E1 -4571.059,E2 -4571.059} C_VEL
LIN {X 0,Y 649.309,Z 995.45,A -85,B 0,C 180,E1 -4572.999,E2 -4572.999} C_VEL
LIN {X 0,Y 648.778,Z 1007.582,A -85,B 0,C 180,E1 -4574.994,E2 -4574.994} C_VEL
LIN {X 0,Y 648.409,Z 1018.409,A -85,B 0,C 180,E1 -4577.057,E2 -4577.057} C_VEL
LIN {X 0,Y 648.153,Z 1027.074,A -85,B 0,C 180,E1 -4579.062,E2 -4579.062} C_VEL
LIN {X 0,Y 648.023,Z 1033.876,A -85,B 0,C 180,E1 -4580.945,E2 -4580.945} C_VEL
LIN {X 0,Y 647.952,Z 1040.172,A -85,B 0,C 180,E1 -4583.176,E2 -4583.176} C_VEL
LIN {X 0,Y 647.916,Z 1044.053,A -85,B 0,C 180,E1 -4585.042,E2 -4585.042} C_VEL
LIN {X 0,Y 647.902,Z 1047.054,A -85,B 0,C 180,E1 -4587.169,E2 -4587.169} C_VEL
LIN {X 0,Y 647.9,Z 1048.294,A -85,B 0,C 180,E1 -4589.204,E2 -4589.204} C_VEL
LIN {X 0,Y 647.914,Z 1048.249,A -85,B 0,C 180,E1 -4591.061,E2 -4591.061} C_VEL
LIN {X 0,Y 647.907,Z 1046.632,A -85,B 0,C 180,E1 -4593.273,E2 -4593.273} C_VEL
LIN {X 0,Y 647.922,Z 1043.896,A -85,B 0,C 180,E1 -4595.135,E2 -4595.135} C_VEL
LIN {X 0,Y 647.965,Z 1039.761,A -85,B 0,C 180,E1 -4597.091,E2 -4597.091} C_VEL
LIN {X 0,Y 648.049,Z 1033.272,A -85,B 0,C 180,E1 -4599.323,E2 -4599.323} C_VEL
LIN {X 0,Y 648.175,Z 1026.366,A -85,B 0,C 180,E1 -4601.208,E2 -4601.208} C_VEL
LIN {X 0,Y 648.45,Z 1016.707,A -85,B 0,C 180,E1 -4603.373,E2 -4603.373} C_VEL
LIN {X 0,Y 648.81,Z 1006.653,A -85,B 0,C 180,E1 -4605.26,E2 -4605.26} C_VEL
LIN {X 0,Y 649.377,Z 993.884,A -85,B 0,C 180,E1 -4607.319,E2 -4607.319} C_VEL
LIN {X 0,Y 650.006,Z 980.858,A -85,B 0,C 180,E1 -4609.126,E2 -4609.126} C_VEL
LIN {X 0,Y 650.879,Z 965.722,A -85,B 0,C 180,E1 -4610.974,E2 -4610.974} C_VEL
LIN {X 0,Y 651.835,Z 949.966,A -85,B 0,C 180,E1 -4612.645,E2 -4612.645} C_VEL
LIN {X 0,Y 653.018,Z 932.128,A -85,B 0,C 180,E1 -4614.324,E2 -4614.324} C_VEL
LIN {X 0,Y 654.227,Z 913.779,A -85,B 0,C 180,E1 -4615.822,E2 -4615.822} C_VEL
LIN {X 0,Y 655.58,Z 894.313,A -85,B 0,C 180,E1 -4617.23,E2 -4617.23} C_VEL
LIN {X 0,Y 656.884,Z 873.852,A -85,B 0,C 180,E1 -4618.503,E2 -4618.503} C_VEL
LIN {X 0,Y 658.327,Z 852.143,A -85,B 0,C 180,E1 -4619.679,E2 -4619.679} C_VEL
LIN {X 0,Y 659.551,Z 830.34,A -85,B 0,C 180,E1 -4620.673,E2 -4620.673} C_VEL
LIN {X 0,Y 660.679,Z 809.675,A -85,B 0,C 180,E1 -4621.475,E2 -4621.475} C_VEL
LIN {X 0,Y 661.819,Z 785.044,A -85,B 0,C 180,E1 -4622.256,E2 -4622.256} C_VEL
LIN {X 0,Y 662.648,Z 764.306,A -85,B 0,C 180,E1 -4622.774,E2 -4622.774} C_VEL
LIN {X 0,Y 663.425,Z 739.334,A -85,B 0,C 180,E1 -4623.243,E2 -4623.243} C_VEL
LIN {X 0,Y 664.288,Z 673.695,A -85,B 0,C 180,E1 -4624.063,E2 -4624.063} C_VEL
LIN {X 0,Y 667.277,Z 426.982,A -85,B 0,C 180,E1 -4627.089,E2 -4627.089} C_VEL
LIN {X 0,Y 667.757,Z 375.753,A -85,B 0,C 180,E1 -4627.739,E2 -4627.739} C_VEL
LIN {X 0,Y 657.165,Z 357.752,A -85,B 0,C 180,E1 -4628.708,E2 -4628.708} C_VEL
LIN {X 0,Y 651.779,Z 348.875,A -85,B 0,C 180,E1 -4629.22,E2 -4629.22} C_VEL
LIN {X 0,Y 648.71,Z 340.427,A -85,B 0,C 180,E1 -4630.228,E2 -4630.228} C_VEL
LIN {X 0,Y 648.719,Z 340.409,A -85,B 0,C 180,E1 -4632.943,E2 -4632.943} C_VEL
LIN {X 0,Y 648.717,Z 340.423,A -85,B 0,C 180,E1 -4636.206,E2 -4636.206} C_VEL
LIN {X 0,Y 648.71,Z 340.394,A -85,B 0,C 180,E1 -4638.957,E2 -4638.957} C_VEL
LIN {X 0,Y 648.736,Z 340.414,A -85,B 0,C 180,E1 -4642.105,E2 -4642.105} C_VEL
LIN {X 0,Y 648.707,Z 340.423,A -85,B 0,C 180,E1 -4644.931,E2 -4644.931} C_VEL
LIN {X 0,Y 648.762,Z 340.413,A -85,B 0,C 180,E1 -4647.982,E2 -4647.982} C_VEL
LIN {X 0,Y 648.703,Z 340.421,A -85,B 0,C 180,E1 -4650.851,E2 -4650.851} C_VEL
LIN {X 0,Y 648.774,Z 340.42,A -85,B 0,C 180,E1 -4653.846,E2 -4653.846} C_VEL
LIN {X 0,Y 648.701,Z 340.414,A -85,B 0,C 180,E1 -4656.855,E2 -4656.855} C_VEL
LIN {X 0,Y 648.753,Z 340.414,A -85,B 0,C 180,E1 -4659.709,E2 -4659.709} C_VEL
LIN {X 0,Y 648.707,Z 340.419,A -85,B 0,C 180,E1 -4662.786,E2 -4662.786} C_VEL
LIN {X 0,Y 648.721,Z 340.413,A -85,B 0,C 180,E1 -4665.54,E2 -4665.54} C_VEL
LIN {X 0,Y 648.719,Z 340.408,A -85,B 0,C 180,E1 -4668.711,E2 -4668.711} C_VEL
LIN {X 0,Y 648.712,Z 340.421,A -85,B 0,C 180,E1 -4671.491,E2 -4671.491} C_VEL
LIN {X 0,Y 648.74,Z 340.415,A -85,B 0,C 180,E1 -4674.605,E2 -4674.605} C_VEL
LIN {X 0,Y 648.703,Z 340.419,A -85,B 0,C 180,E1 -4677.438,E2 -4677.438} C_VEL
LIN {X 0,Y 648.773,Z 340.417,A -85,B 0,C 180,E1 -4680.442,E2 -4680.442} C_VEL
LIN {X 0,Y 648.7,Z 340.408,A -85,B 0,C 180,E1 -4683.358,E2 -4683.358} C_VEL
LIN {X 0,Y 648.767,Z 340.416,A -85,B 0,C 180,E1 -4686.282,E2 -4686.282} C_VEL
LIN {X 0,Y 648.704,Z 340.418,A -85,B 0,C 180,E1 -4689.314,E2 -4689.314} C_VEL
LIN {X 0,Y 648.745,Z 340.413,A -85,B 0,C 180,E1 -4692.19,E2 -4692.19} C_VEL
LIN {X 0,Y 648.709,Z 340.417,A -85,B 0,C 180,E1 -4695.282,E2 -4695.282} C_VEL
LIN {X 0,Y 648.718,Z 340.418,A -85,B 0,C 180,E1 -4698.048,E2 -4698.048} C_VEL
LIN {X 0,Y 648.721,Z 340.414,A -85,B 0,C 180,E1 -4701.236,E2 -4701.236} C_VEL
LIN {X 0,Y 648.706,Z 340.419,A -85,B 0,C 180,E1 -4703.932,E2 -4703.932} C_VEL
LIN {X 0,Y 648.754,Z 340.413,A -85,B 0,C 180,E1 -4707.044,E2 -4707.044} C_VEL
LIN {X 0,Y 648.701,Z 340.422,A -85,B 0,C 180,E1 -4709.859,E2 -4709.859} C_VEL
LIN {X 0,Y 648.773,Z 340.42,A -85,B 0,C 180,E1 -4712.854,E2 -4712.854} C_VEL
LIN {X 0,Y 648.701,Z 340.422,A -85,B 0,C 180,E1 -4715.854,E2 -4715.854} C_VEL
LIN {X 0,Y 648.761,Z 340.419,A -85,B 0,C 180,E1 -4718.752,E2 -4718.752} C_VEL
LIN {X 0,Y 648.706,Z 340.409,A -85,B 0,C 180,E1 -4721.753,E2 -4721.753} C_VEL
LIN {X 0,Y 648.722,Z 340.419,A -85,B 0,C 180,E1 -4724.532,E2 -4724.532} C_VEL
LIN {X 0,Y 648.734,Z 340.514,A -85,B 0,C 180,E1 -4727.659,E2 -4727.659} C_VEL
LIN {X 0,Y 657.755,Z 363.85,A -85,B 0,C 180,E1 -4730.282,E2 -4730.282} C_VEL
LIN {X 0,Y 661.542,Z 374.764,A -85,B 0,C 180,E1 -4731.424,E2 -4731.424} C_VEL
LIN {X 0,Y 661.641,Z 376.522,A -85,B 0,C 180,E1 -4731.528,E2 -4731.528} C_VEL
LIN {X 0,Y 667.866,Z 402.911,A -85,B 0,C 180,E1 -4732.3,E2 -4732.3} C_VEL
LIN {X 0,Y 664.638,Z 669.09,A -85,B 0,C 180,E1 -4735.568,E2 -4735.568} C_VEL
LIN {X 0,Y 663.414,Z 767.864,A -85,B 0,C 180,E1 -4736.785,E2 -4736.785} C_VEL
LIN {X 0,Y 662.659,Z 793.277,A -85,B 0,C 180,E1 -4737.252,E2 -4737.252} C_VEL
LIN {X 0,Y 661.842,Z 814.057,A -85,B 0,C 180,E1 -4737.765,E2 -4737.765} C_VEL
LIN {X 0,Y 660.815,Z 837.254,A -85,B 0,C 180,E1 -4738.481,E2 -4738.481} C_VEL
LIN {X 0,Y 659.604,Z 859.333,A -85,B 0,C 180,E1 -4739.33,E2 -4739.33} C_VEL
LIN {X 0,Y 658.379,Z 881.27,A -85,B 0,C 180,E1 -4740.324,E2 -4740.324} C_VEL
LIN {X 0,Y 656.935,Z 903.116,A -85,B 0,C 180,E1 -4741.5,E2 -4741.5} C_VEL
LIN {X 0,Y 655.616,Z 923.648,A -85,B 0,C 180,E1 -4742.772,E2 -4742.772} C_VEL
LIN {X 0,Y 654.268,Z 943.216,A -85,B 0,C 180,E1 -4744.179,E2 -4744.179} C_VEL
LIN {X 0,Y 653.066,Z 961.202,A -85,B 0,C 180,E1 -4745.643,E2 -4745.643} C_VEL
LIN {X 0,Y 651.926,Z 978.602,A -85,B 0,C 180,E1 -4747.263,E2 -4747.263} C_VEL
LIN {X 0,Y 650.992,Z 993.628,A -85,B 0,C 180,E1 -4748.842,E2 -4748.842} C_VEL
LIN {X 0,Y 650.059,Z 1010.028,A -85,B 0,C 180,E1 -4750.81,E2 -4750.81} C_VEL
LIN {X 0,Y 649.428,Z 1022.519,A -85,B 0,C 180,E1 -4752.528,E2 -4752.528} C_VEL
LIN {X 0,Y 648.846,Z 1035.767,A -85,B 0,C 180,E1 -4754.63,E2 -4754.63} C_VEL
LIN {X 0,Y 648.494,Z 1045.562,A -85,B 0,C 180,E1 -4756.446,E2 -4756.446} C_VEL
LIN {X 0,Y 648.208,Z 1055.478,A -85,B 0,C 180,E1 -4758.612,E2 -4758.612} C_VEL
LIN {X 0,Y 648.055,Z 1062.514,A -85,B 0,C 180,E1 -4760.497,E2 -4760.497} C_VEL
LIN {X 0,Y 647.954,Z 1068.761,A -85,B 0,C 180,E1 -4762.552,E2 -4762.552} C_VEL
LIN {X 0,Y 647.924,Z 1073.496,A -85,B 0,C 180,E1 -4764.687,E2 -4764.687} C_VEL
LIN {X 0,Y 647.913,Z 1076.35,A -85,B 0,C 180,E1 -4766.549,E2 -4766.549} C_VEL
LIN {X 0,Y 647.905,Z 1078.192,A -85,B 0,C 180,E1 -4768.762,E2 -4768.762} C_VEL
LIN {X 0,Y 647.897,Z 1078.328,A -85,B 0,C 180,E1 -4770.707,E2 -4770.707} C_VEL
LIN {X 0,Y 647.907,Z 1077.157,A -85,B 0,C 180,E1 -4772.742,E2 -4772.742} C_VEL
LIN {X 0,Y 647.925,Z 1074.133,A -85,B 0,C 180,E1 -4774.958,E2 -4774.958} C_VEL
LIN {X 0,Y 647.94,Z 1070.276,A -85,B 0,C 180,E1 -4776.824,E2 -4776.824} C_VEL
LIN {X 0,Y 648.021,Z 1064.006,A -85,B 0,C 180,E1 -4779.062,E2 -4779.062} C_VEL
LIN {X 0,Y 648.158,Z 1057.25,A -85,B 0,C 180,E1 -4780.938,E2 -4780.938} C_VEL
LIN {X 0,Y 648.402,Z 1048.623,A -85,B 0,C 180,E1 -4782.941,E2 -4782.941} C_VEL
LIN {X 0,Y 648.764,Z 1037.836,A -85,B 0,C 180,E1 -4785.006,E2 -4785.006} C_VEL
LIN {X 0,Y 649.259,Z 1026.235,A -85,B 0,C 180,E1 -4786.922,E2 -4786.922} C_VEL
LIN {X 0,Y 649.924,Z 1012.348,A -85,B 0,C 180,E1 -4788.886,E2 -4788.886} C_VEL
LIN {X 0,Y 650.774,Z 997.755,A -85,B 0,C 180,E1 -4790.694,E2 -4790.694} C_VEL
LIN {X 0,Y 651.742,Z 981.382,A -85,B 0,C 180,E1 -4792.458,E2 -4792.458} C_VEL
LIN {X 0,Y 652.838,Z 964.772,A -85,B 0,C 180,E1 -4794.042,E2 -4794.042} C_VEL
LIN {X 0,Y 654.088,Z 945.649,A -85,B 0,C 180,E1 -4795.634,E2 -4795.634} C_VEL
LIN {X 0,Y 655.324,Z 927.728,A -85,B 0,C 180,E1 -4796.947,E2 -4796.947} C_VEL
LIN {X 0,Y 656.777,Z 905.547,A -85,B 0,C 180,E1 -4798.359,E2 -4798.359} C_VEL
LIN {X 0,Y 658.052,Z 885.846,A -85,B 0,C 180,E1 -4799.442,E2 -4799.442} C_VEL
LIN {X 0,Y 659.456,Z 862.308,A -85,B 0,C 180,E1 -4800.545,E2 -4800.545} C_VEL
LIN {X 0,Y 660.538,Z 842.396,A -85,B 0,C 180,E1 -4801.33,E2 -4801.33} C_VEL
LIN {X 0,Y 661.642,Z 818.854,A -85,B 0,C 180,E1 -4802.105,E2 -4802.105} C_VEL
LIN {X 0,Y 662.54,Z 796.098,A -85,B 0,C 180,E1 -4802.685,E2 -4802.685} C_VEL
LIN {X 0,Y 663.334,Z 772.6,A -85,B 0,C 180,E1 -4803.144,E2 -4803.144} C_VEL
LIN {X 0,Y 663.909,Z 733.544,A -85,B 0,C 180,E1 -4803.652,E2 -4803.652} C_VEL
LIN {X 0,Y 666.861,Z 482.204,A -85,B 0,C 180,E1 -4806.718,E2 -4806.718} C_VEL
LIN {X 0,Y 667.697,Z 401.372,A -85,B 0,C 180,E1 -4807.732,E2 -4807.732} C_VEL
LIN {X 0,Y 661.512,Z 375.525,A -85,B 0,C 180,E1 -4808.517,E2 -4808.517} C_VEL
LIN {X 0,Y 661.212,Z 373.348,A -85,B 0,C 180,E1 -4808.712,E2 -4808.712} C_VEL
LIN {X 0,Y 653.404,Z 352.635,A -85,B 0,C 180,E1 -4810.957,E2 -4810.957} C_VEL
LIN {X 0,Y 648.725,Z 340.419,A -85,B 0,C 180,E1 -4812.372,E2 -4812.372} C_VEL
LIN {X 0,Y 648.714,Z 340.42,A -85,B 0,C 180,E1 -4815.591,E2 -4815.591} C_VEL
LIN {X 0,Y 648.716,Z 340.417,A -85,B 0,C 180,E1 -4818.378,E2 -4818.378} C_VEL
LIN {X 0,Y 648.723,Z 340.422,A -85,B 0,C 180,E1 -4821.599,E2 -4821.599} C_VEL
LIN {X 0,Y 648.706,Z 340.385,A -85,B 0,C 180,E1 -4824.364,E2 -4824.364} C_VEL
LIN {X 0,Y 648.747,Z 340.419,A -85,B 0,C 180,E1 -4827.466,E2 -4827.466} C_VEL
LIN {X 0,Y 648.704,Z 340.419,A -85,B 0,C 180,E1 -4830.243,E2 -4830.243} C_VEL
LIN {X 0,Y 648.774,Z 340.409,A -85,B 0,C 180,E1 -4833.17,E2 -4833.17} C_VEL
LIN {X 0,Y 648.704,Z 340.416,A -85,B 0,C 180,E1 -4836.182,E2 -4836.182} C_VEL
LIN {X 0,Y 648.742,Z 340.417,A -85,B 0,C 180,E1 -4838.954,E2 -4838.954} C_VEL
LIN {X 0,Y 648.716,Z 340.421,A -85,B 0,C 180,E1 -4842.045,E2 -4842.045} C_VEL
LIN {X 0,Y 648.717,Z 340.413,A -85,B 0,C 180,E1 -4844.81,E2 -4844.81} C_VEL
LIN {X 0,Y 648.729,Z 340.412,A -85,B 0,C 180,E1 -4847.99,E2 -4847.99} C_VEL
LIN {X 0,Y 648.709,Z 340.419,A -85,B 0,C 180,E1 -4850.776,E2 -4850.776} C_VEL
LIN {X 0,Y 648.754,Z 340.416,A -85,B 0,C 180,E1 -4853.895,E2 -4853.895} C_VEL
LIN {X 0,Y 648.704,Z 340.413,A -85,B 0,C 180,E1 -4856.731,E2 -4856.731} C_VEL
LIN {X 0,Y 648.777,Z 340.418,A -85,B 0,C 180,E1 -4859.735,E2 -4859.735} C_VEL
LIN {X 0,Y 648.704,Z 340.415,A -85,B 0,C 180,E1 -4862.739,E2 -4862.739} C_VEL
LIN {X 0,Y 648.77,Z 340.416,A -85,B 0,C 180,E1 -4865.661,E2 -4865.661} C_VEL
LIN {X 0,Y 648.709,Z 340.421,A -85,B 0,C 180,E1 -4868.688,E2 -4868.688} C_VEL
LIN {X 0,Y 648.747,Z 340.407,A -85,B 0,C 180,E1 -4871.558,E2 -4871.558} C_VEL
LIN {X 0,Y 648.716,Z 340.416,A -85,B 0,C 180,E1 -4874.642,E2 -4874.642} C_VEL
LIN {X 0,Y 648.731,Z 340.416,A -85,B 0,C 180,E1 -4877.491,E2 -4877.491} C_VEL
LIN {X 0,Y 648.723,Z 340.42,A -85,B 0,C 180,E1 -4880.678,E2 -4880.678} C_VEL
LIN {X 0,Y 648.723,Z 340.414,A -85,B 0,C 180,E1 -4883.497,E2 -4883.497} C_VEL
LIN {X 0,Y 648.725,Z 340.417,A -85,B 0,C 180,E1 -4886.748,E2 -4886.748} C_VEL
LIN {X 0,Y 648.721,Z 340.418,A -85,B 0,C 180,E1 -4889.553,E2 -4889.553} C_VEL
LIN {X 0,Y 648.736,Z 340.423,A -85,B 0,C 180,E1 -4892.751,E2 -4892.751} C_VEL
LIN {X 0,Y 648.714,Z 340.418,A -85,B 0,C 180,E1 -4895.528,E2 -4895.528} C_VEL
LIN {X 0,Y 648.765,Z 340.418,A -85,B 0,C 180,E1 -4898.623,E2 -4898.623} C_VEL
LIN {X 0,Y 648.711,Z 340.422,A -85,B 0,C 180,E1 -4901.513,E2 -4901.513} C_VEL
LIN {X 0,Y 648.772,Z 340.416,A -85,B 0,C 180,E1 -4902.432,E2 -4902.432} C_VEL
LIN {X 0,Y 647.759,Z 340.54,A -85,B 0,C 180,E1 -4903.112,E2 -4903.112} C_VEL
LIN {X 0,Y 641.298,Z 341.345,A -85,B 0,C 180,E1 -4905.019,E2 -4905.019} C_VEL
LIN {X 0,Y 640.771,Z 341.41,A -85,B 0,C 180,E1 -4905.516,E2 -4905.516} C_VEL
LIN {X 0,Y 640.837,Z 341.405,A -85,B 0,C 180,E1 -4908.581,E2 -4908.581} C_VEL
LIN {X 0,Y 640.797,Z 341.565,A -85,B 0,C 180,E1 -4909.347,E2 -4909.347} C_VEL
LIN {X 0,Y 643.874,Z 349.579,A -85,B 0,C 180,E1 -4910.307,E2 -4910.307} C_VEL
LIN {X 0,Y 658.732,Z 374.124,A -85,B 0,C 180,E1 -4911.716,E2 -4911.716} C_VEL
LIN {X 0,Y 661.55,Z 379.488,A -85,B 0,C 180,E1 -4911.983,E2 -4911.983} C_VEL
LIN {X 0,Y 658.32,Z 622.133,A -85,B 0,C 180,E1 -4915.002,E2 -4915.002} C_VEL
LIN {X 0,Y 656.759,Z 738.173,A -85,B 0,C 180,E1 -4916.444,E2 -4916.444} C_VEL
LIN {X 0,Y 655.957,Z 763.515,A -85,B 0,C 180,E1 -4916.914,E2 -4916.914} C_VEL
LIN {X 0,Y 655.089,Z 784.009,A -85,B 0,C 180,E1 -4917.425,E2 -4917.425} C_VEL
LIN {X 0,Y 654.023,Z 806.302,A -85,B 0,C 180,E1 -4918.115,E2 -4918.115} C_VEL
LIN {X 0,Y 652.683,Z 828.427,A -85,B 0,C 180,E1 -4918.969,E2 -4918.969} C_VEL
LIN {X 0,Y 651.407,Z 849.388,A -85,B 0,C 180,E1 -4919.923,E2 -4919.923} C_VEL
LIN {X 0,Y 649.873,Z 871.573,A -85,B 0,C 180,E1 -4921.111,E2 -4921.111} C_VEL
LIN {X 0,Y 648.485,Z 890.786,A -85,B 0,C 180,E1 -4922.298,E2 -4922.298} C_VEL
LIN {X 0,Y 646.954,Z 912.02,A -85,B 0,C 180,E1 -4923.814,E2 -4923.814} C_VEL
LIN {X 0,Y 645.715,Z 928.887,A -85,B 0,C 180,E1 -4925.188,E2 -4925.188} C_VEL
LIN {X 0,Y 644.343,Z 948.172,A -85,B 0,C 180,E1 -4926.98,E2 -4926.98} C_VEL
LIN {X 0,Y 643.311,Z 963.392,A -85,B 0,C 180,E1 -4928.595,E2 -4928.595} C_VEL
LIN {X 0,Y 642.27,Z 980.198,A -85,B 0,C 180,E1 -4930.636,E2 -4930.636} C_VEL
LIN {X 0,Y 641.56,Z 992.85,A -85,B 0,C 180,E1 -4932.401,E2 -4932.401} C_VEL
LIN {X 0,Y 640.926,Z 1006.041,A -85,B 0,C 180,E1 -4934.528,E2 -4934.528} C_VEL
LIN {X 0,Y 640.542,Z 1015.799,A -85,B 0,C 180,E1 -4936.366,E2 -4936.366} C_VEL
LIN {X 0,Y 640.231,Z 1025.658,A -85,B 0,C 180,E1 -4938.56,E2 -4938.56} C_VEL
LIN {X 0,Y 640.065,Z 1032.666,A -85,B 0,C 180,E1 -4940.469,E2 -4940.469} C_VEL
LIN {X 0,Y 639.958,Z 1038.889,A -85,B 0,C 180,E1 -4942.549,E2 -4942.549} C_VEL
LIN {X 0,Y 639.919,Z 1043.575,A -85,B 0,C 180,E1 -4944.711,E2 -4944.711} C_VEL
LIN {X 0,Y 639.912,Z 1046.406,A -85,B 0,C 180,E1 -4946.596,E2 -4946.596} C_VEL
LIN {X 0,Y 639.91,Z 1048.203,A -85,B 0,C 180,E1 -4948.836,E2 -4948.836} C_VEL
LIN {X 0,Y 639.901,Z 1048.316,A -85,B 0,C 180,E1 -4950.806,E2 -4950.806} C_VEL
LIN {X 0,Y 639.903,Z 1047.123,A -85,B 0,C 180,E1 -4952.866,E2 -4952.866} C_VEL
LIN {X 0,Y 639.921,Z 1044.214,A -85,B 0,C 180,E1 -4955.02,E2 -4955.02} C_VEL
LIN {X 0,Y 639.952,Z 1040.379,A -85,B 0,C 180,E1 -4956.91,E2 -4956.91} C_VEL
LIN {X 0,Y 640.039,Z 1034.179,A -85,B 0,C 180,E1 -4959.169,E2 -4959.169} C_VEL
LIN {X 0,Y 640.174,Z 1027.425,A -85,B 0,C 180,E1 -4961.076,E2 -4961.076} C_VEL
LIN {X 0,Y 640.433,Z 1019.14,A -85,B 0,C 180,E1 -4963.033,E2 -4963.033} C_VEL
LIN {X 0,Y 640.828,Z 1008.595,A -85,B 0,C 180,E1 -4965.104,E2 -4965.104} C_VEL
LIN {X 0,Y 641.326,Z 997.671,A -85,B 0,C 180,E1 -4966.951,E2 -4966.951} C_VEL
LIN {X 0,Y 642.076,Z 983.29,A -85,B 0,C 180,E1 -4969.043,E2 -4969.043} C_VEL
LIN {X 0,Y 642.922,Z 969.672,A -85,B 0,C 180,E1 -4970.768,E2 -4970.768} C_VEL
LIN {X 0,Y 644.028,Z 952.737,A -85,B 0,C 180,E1 -4972.646,E2 -4972.646} C_VEL
LIN {X 0,Y 645.111,Z 937.265,A -85,B 0,C 180,E1 -4974.154,E2 -4974.154} C_VEL
LIN {X 0,Y 646.542,Z 917.419,A -85,B 0,C 180,E1 -4975.857,E2 -4975.857} C_VEL
LIN {X 0,Y 647.857,Z 899.669,A -85,B 0,C 180,E1 -4977.183,E2 -4977.183} C_VEL
LIN {X 0,Y 649.378,Z 878.709,A -85,B 0,C 180,E1 -4978.561,E2 -4978.561} C_VEL
LIN {X 0,Y 650.764,Z 858.438,A -85,B 0,C 180,E1 -4979.704,E2 -4979.704} C_VEL
LIN {X 0,Y 652.274,Z 836.018,A -85,B 0,C 180,E1 -4980.797,E2 -4980.797} C_VEL
LIN {X 0,Y 653.52,Z 814.946,A -85,B 0,C 180,E1 -4981.654,E2 -4981.654} C_VEL
LIN {X 0,Y 654.602,Z 794.419,A -85,B 0,C 180,E1 -4982.36,E2 -4982.36} C_VEL
LIN {X 0,Y 655.712,Z 769.173,A -85,B 0,C 180,E1 -4983.048,E2 -4983.048} C_VEL
LIN {X 0,Y 656.49,Z 747.652,A -85,B 0,C 180,E1 -4983.49,E2 -4983.49} C_VEL
LIN {X 0,Y 657.13,Z 717.059,A -85,B 0,C 180,E1 -4983.926,E2 -4983.926} C_VEL
LIN {X 0,Y 660.438,Z 462.322,A -85,B 0,C 180,E1 -4987.067,E2 -4987.067} C_VEL
LIN {X 0,Y 661.447,Z 378.914,A -85,B 0,C 180,E1 -4988.122,E2 -4988.122} C_VEL
LIN {X 0,Y 651.495,Z 362.073,A -85,B 0,C 180,E1 -4989.05,E2 -4989.05} C_VEL
LIN {X 0,Y 643.668,Z 349.163,A -85,B 0,C 180,E1 -4989.81,E2 -4989.81} C_VEL
LIN {X 0,Y 640.774,Z 341.41,A -85,B 0,C 180,E1 -4990.795,E2 -4990.795} C_VEL
LIN {X 0,Y 640.794,Z 341.381,A -85,B 0,C 180,E1 -4993.977,E2 -4993.977} C_VEL
LIN {X 0,Y 640.768,Z 341.415,A -85,B 0,C 180,E1 -4996.78,E2 -4996.78} C_VEL
LIN {X 0,Y 640.822,Z 341.391,A -85,B 0,C 180,E1 -4999.878,E2 -4999.878} C_VEL
LIN {X 0,Y 640.764,Z 341.406,A -85,B 0,C 180,E1 -5002.738,E2 -5002.738} C_VEL
LIN {X 0,Y 640.834,Z 341.4,A -85,B 0,C 180,E1 -5005.787,E2 -5005.787} C_VEL
LIN {X 0,Y 640.763,Z 341.405,A -85,B 0,C 180,E1 -5008.797,E2 -5008.797} C_VEL
LIN {X 0,Y 640.831,Z 341.402,A -85,B 0,C 180,E1 -5011.684,E2 -5011.684} C_VEL
LIN {X 0,Y 640.767,Z 341.409,A -85,B 0,C 180,E1 -5014.687,E2 -5014.687} C_VEL
LIN {X 0,Y 640.798,Z 341.406,A -85,B 0,C 180,E1 -5017.524,E2 -5017.524} C_VEL
LIN {X 0,Y 640.773,Z 341.401,A -85,B 0,C 180,E1 -5020.682,E2 -5020.682} C_VEL
LIN {X 0,Y 640.784,Z 341.412,A -85,B 0,C 180,E1 -5023.501,E2 -5023.501} C_VEL
LIN {X 0,Y 640.776,Z 341.408,A -85,B 0,C 180,E1 -5026.739,E2 -5026.739} C_VEL
LIN {X 0,Y 640.78,Z 341.399,A -85,B 0,C 180,E1 -5029.571,E2 -5029.571} C_VEL
LIN {X 0,Y 640.775,Z 341.402,A -85,B 0,C 180,E1 -5032.829,E2 -5032.829} C_VEL
LIN {X 0,Y 640.776,Z 341.409,A -85,B 0,C 180,E1 -5035.615,E2 -5035.615} C_VEL
LIN {X 0,Y 640.783,Z 341.4,A -85,B 0,C 180,E1 -5038.838,E2 -5038.838} C_VEL
LIN {X 0,Y 640.766,Z 341.41,A -85,B 0,C 180,E1 -5041.52,E2 -5041.52} C_VEL
LIN {X 0,Y 640.826,Z 341.406,A -85,B 0,C 180,E1 -5044.564,E2 -5044.564} C_VEL
LIN {X 0,Y 640.76,Z 341.402,A -85,B 0,C 180,E1 -5047.442,E2 -5047.442} C_VEL
LIN {X 0,Y 640.832,Z 341.406,A -85,B 0,C 180,E1 -5050.428,E2 -5050.428} C_VEL
LIN {X 0,Y 640.762,Z 341.406,A -85,B 0,C 180,E1 -5053.445,E2 -5053.445} C_VEL
LIN {X 0,Y 640.816,Z 341.4,A -85,B 0,C 180,E1 -5056.34,E2 -5056.34} C_VEL
LIN {X 0,Y 640.767,Z 341.406,A -85,B 0,C 180,E1 -5059.413,E2 -5059.413} C_VEL
LIN {X 0,Y 640.787,Z 341.407,A -85,B 0,C 180,E1 -5062.186,E2 -5062.186} C_VEL
LIN {X 0,Y 640.774,Z 341.406,A -85,B 0,C 180,E1 -5065.412,E2 -5065.412} C_VEL
LIN {X 0,Y 640.775,Z 341.405,A -85,B 0,C 180,E1 -5068.158,E2 -5068.158} C_VEL
LIN {X 0,Y 640.779,Z 341.404,A -85,B 0,C 180,E1 -5071.4,E2 -5071.4} C_VEL
LIN {X 0,Y 640.772,Z 341.409,A -85,B 0,C 180,E1 -5074.204,E2 -5074.204} C_VEL
LIN {X 0,Y 640.79,Z 341.407,A -85,B 0,C 180,E1 -5077.416,E2 -5077.416} C_VEL
LIN {X 0,Y 640.762,Z 341.394,A -85,B 0,C 180,E1 -5080.127,E2 -5080.127} C_VEL
LIN {X 0,Y 640.832,Z 341.407,A -85,B 0,C 180,E1 -5083.111,E2 -5083.111} C_VEL
LIN {X 0,Y 640.763,Z 341.408,A -85,B 0,C 180,E1 -5086.02,E2 -5086.02} C_VEL
LIN {X 0,Y 640.864,Z 341.634,A -85,B 0,C 180,E1 -5087.136,E2 -5087.136} C_VEL
LIN {X 0,Y 648.814,Z 362.226,A -85,B 0,C 180,E1 -5089.512,E2 -5089.512} C_VEL
LIN {X 0,Y 654.007,Z 376.022,A -85,B 0,C 180,E1 -5090.991,E2 -5090.991} C_VEL
LIN {X 0,Y 655.595,Z 379.447,A -85,B 0,C 180,E1 -5091.15,E2 -5091.15} C_VEL
LIN {X 0,Y 661.496,Z 404.628,A -85,B 0,C 180,E1 -5091.898,E2 -5091.898} C_VEL
LIN {X 0,Y 657.99,Z 671.808,A -85,B 0,C 180,E1 -5095.209,E2 -5095.209} C_VEL
LIN {X 0,Y 656.701,Z 767.711,A -85,B 0,C 180,E1 -5096.401,E2 -5096.401} C_VEL
LIN {X 0,Y 655.893,Z 793.061,A -85,B 0,C 180,E1 -5096.871,E2 -5096.871} C_VEL
LIN {X 0,Y 655.031,Z 813.514,A -85,B 0,C 180,E1 -5097.379,E2 -5097.379} C_VEL
LIN {X 0,Y 653.953,Z 836.429,A -85,B 0,C 180,E1 -5098.086,E2 -5098.086} C_VEL
LIN {X 0,Y 652.609,Z 859.258,A -85,B 0,C 180,E1 -5098.965,E2 -5098.965} C_VEL
LIN {X 0,Y 651.357,Z 880.27,A -85,B 0,C 180,E1 -5099.92,E2 -5099.92} C_VEL
LIN {X 0,Y 649.815,Z 902.323,A -85,B 0,C 180,E1 -5101.109,E2 -5101.109} C_VEL
LIN {X 0,Y 648.443,Z 921.454,A -85,B 0,C 180,E1 -5102.296,E2 -5102.296} C_VEL
LIN {X 0,Y 646.957,Z 941.997,A -85,B 0,C 180,E1 -5103.767,E2 -5103.767} C_VEL
LIN {X 0,Y 645.698,Z 959.035,A -85,B 0,C 180,E1 -5105.155,E2 -5105.155} C_VEL
LIN {X 0,Y 644.314,Z 978.601,A -85,B 0,C 180,E1 -5106.979,E2 -5106.979} C_VEL
LIN {X 0,Y 643.283,Z 993.855,A -85,B 0,C 180,E1 -5108.601,E2 -5108.601} C_VEL
LIN {X 0,Y 642.297,Z 1009.818,A -85,B 0,C 180,E1 -5110.54,E2 -5110.54} C_VEL
LIN {X 0,Y 641.577,Z 1022.517,A -85,B 0,C 180,E1 -5112.308,E2 -5112.308} C_VEL
LIN {X 0,Y 640.946,Z 1035.768,A -85,B 0,C 180,E1 -5114.435,E2 -5114.435} C_VEL
LIN {X 0,Y 640.557,Z 1045.561,A -85,B 0,C 180,E1 -5116.275,E2 -5116.275} C_VEL
LIN {X 0,Y 640.244,Z 1055.479,A -85,B 0,C 180,E1 -5118.469,E2 -5118.469} C_VEL
LIN {X 0,Y 640.064,Z 1062.513,A -85,B 0,C 180,E1 -5120.378,E2 -5120.378} C_VEL
LIN {X 0,Y 639.958,Z 1068.507,A -85,B 0,C 180,E1 -5122.368,E2 -5122.368} C_VEL
LIN {X 0,Y 639.926,Z 1073.336,A -85,B 0,C 180,E1 -5124.531,E2 -5124.531} C_VEL
LIN {X 0,Y 639.908,Z 1076.238,A -85,B 0,C 180,E1 -5126.416,E2 -5126.416} C_VEL
LIN {X 0,Y 639.894,Z 1078.146,A -85,B 0,C 180,E1 -5128.567,E2 -5128.567} C_VEL
LIN {X 0,Y 639.894,Z 1078.35,A -85,B 0,C 180,E1 -5130.627,E2 -5130.627} C_VEL
LIN {X 0,Y 639.907,Z 1077.293,A -85,B 0,C 180,E1 -5132.597,E2 -5132.597} C_VEL
LIN {X 0,Y 639.924,Z 1074.451,A -85,B 0,C 180,E1 -5134.84,E2 -5134.84} C_VEL
LIN {X 0,Y 639.935,Z 1070.689,A -85,B 0,C 180,E1 -5136.73,E2 -5136.73} C_VEL
LIN {X 0,Y 640.008,Z 1065.202,A -85,B 0,C 180,E1 -5138.807,E2 -5138.807} C_VEL
LIN {X 0,Y 640.169,Z 1057.956,A -85,B 0,C 180,E1 -5140.894,E2 -5140.894} C_VEL
LIN {X 0,Y 640.404,Z 1049.938,A -85,B 0,C 180,E1 -5142.809,E2 -5142.809} C_VEL
LIN {X 0,Y 640.813,Z 1038.847,A -85,B 0,C 180,E1 -5145.015,E2 -5145.015} C_VEL
LIN {X 0,Y 641.3,Z 1027.973,A -85,B 0,C 180,E1 -5146.858,E2 -5146.858} C_VEL
LIN {X 0,Y 642.038,Z 1014.023,A -85,B 0,C 180,E1 -5148.901,E2 -5148.901} C_VEL
LIN {X 0,Y 642.842,Z 1000.85,A -85,B 0,C 180,E1 -5150.581,E2 -5150.581} C_VEL
LIN {X 0,Y 643.933,Z 984.158,A -85,B 0,C 180,E1 -5152.457,E2 -5152.457} C_VEL
LIN {X 0,Y 645.033,Z 968.319,A -85,B 0,C 180,E1 -5154.011,E2 -5154.011} C_VEL
LIN {X 0,Y 646.361,Z 950.194,A -85,B 0,C 180,E1 -5155.594,E2 -5155.594} C_VEL
LIN {X 0,Y 647.745,Z 931.054,A -85,B 0,C 180,E1 -5157.04,E2 -5157.04} C_VEL
LIN {X 0,Y 649.228,Z 911.162,A -85,B 0,C 180,E1 -5158.368,E2 -5158.368} C_VEL
LIN {X 0,Y 650.633,Z 890.294,A -85,B 0,C 180,E1 -5159.561,E2 -5159.561} C_VEL
LIN {X 0,Y 651.972,Z 870.218,A -85,B 0,C 180,E1 -5160.557,E2 -5160.557} C_VEL
LIN {X 0,Y 653.35,Z 847.075,A -85,B 0,C 180,E1 -5161.522,E2 -5161.522} C_VEL
LIN {X 0,Y 654.406,Z 826.844,A -85,B 0,C 180,E1 -5162.225,E2 -5162.225} C_VEL
LIN {X 0,Y 655.479,Z 803.659,A -85,B 0,C 180,E1 -5162.888,E2 -5162.888} C_VEL
LIN {X 0,Y 656.329,Z 779.732,A -85,B 0,C 180,E1 -5163.397,E2 -5163.397} C_VEL
LIN {X 0,Y 656.971,Z 755.127,A -85,B 0,C 180,E1 -5163.775,E2 -5163.775} C_VEL
LIN {X 0,Y 660.104,Z 506.214,A -85,B 0,C 180,E1 -5166.835,E2 -5166.835} C_VEL
LIN {X 0,Y 661.336,Z 403.157,A -85,B 0,C 180,E1 -5168.133,E2 -5168.133} C_VEL
LIN {X 0,Y 655.032,Z 377.89,A -85,B 0,C 180,E1 -5168.911,E2 -5168.911} C_VEL
LIN {X 0,Y 653.657,Z 375.258,A -85,B 0,C 180,E1 -5169.067,E2 -5169.067} C_VEL
LIN {X 0,Y 645.948,Z 354.603,A -85,B 0,C 180,E1 -5171.344,E2 -5171.344} C_VEL
LIN {X 0,Y 640.833,Z 341.409,A -85,B 0,C 180,E1 -5172.908,E2 -5172.908} C_VEL
LIN {X 0,Y 640.764,Z 341.41,A -85,B 0,C 180,E1 -5175.895,E2 -5175.895} C_VEL
LIN {X 0,Y 640.836,Z 341.405,A -85,B 0,C 180,E1 -5178.905,E2 -5178.905} C_VEL
LIN {X 0,Y 640.764,Z 341.409,A -85,B 0,C 180,E1 -5181.947,E2 -5181.947} C_VEL
LIN {X 0,Y 640.814,Z 341.369,A -85,B 0,C 180,E1 -5184.847,E2 -5184.847} C_VEL
LIN {X 0,Y 640.768,Z 341.405,A -85,B 0,C 180,E1 -5187.922,E2 -5187.922} C_VEL
LIN {X 0,Y 640.792,Z 341.405,A -85,B 0,C 180,E1 -5190.722,E2 -5190.722} C_VEL
LIN {X 0,Y 640.78,Z 341.41,A -85,B 0,C 180,E1 -5193.893,E2 -5193.893} C_VEL
LIN {X 0,Y 640.777,Z 341.402,A -85,B 0,C 180,E1 -5196.65,E2 -5196.65} C_VEL
LIN {X 0,Y 640.792,Z 341.403,A -85,B 0,C 180,E1 -5199.827,E2 -5199.827} C_VEL
LIN {X 0,Y 640.772,Z 341.407,A -85,B 0,C 180,E1 -5202.66,E2 -5202.66} C_VEL
LIN {X 0,Y 640.806,Z 341.412,A -85,B 0,C 180,E1 -5205.819,E2 -5205.819} C_VEL
LIN {X 0,Y 640.767,Z 341.4,A -85,B 0,C 180,E1 -5208.661,E2 -5208.661} C_VEL
LIN {X 0,Y 640.828,Z 341.401,A -85,B 0,C 180,E1 -5211.747,E2 -5211.747} C_VEL
LIN {X 0,Y 640.766,Z 341.409,A -85,B 0,C 180,E1 -5214.628,E2 -5214.628} C_VEL
LIN {X 0,Y 640.83,Z 341.396,A -85,B 0,C 180,E1 -5217.586,E2 -5217.586} C_VEL
LIN {X 0,Y 640.769,Z 341.406,A -85,B 0,C 180,E1 -5220.626,E2 -5220.626} C_VEL
LIN {X 0,Y 640.824,Z 341.4,A -85,B 0,C 180,E1 -5223.578,E2 -5223.578} C_VEL
LIN {X 0,Y 640.769,Z 341.399,A -85,B 0,C 180,E1 -5226.631,E2 -5226.631} C_VEL
LIN {X 0,Y 640.81,Z 341.406,A -85,B 0,C 180,E1 -5229.52,E2 -5229.52} C_VEL
LIN {X 0,Y 640.778,Z 341.41,A -85,B 0,C 180,E1 -5232.619,E2 -5232.619} C_VEL
LIN {X 0,Y 640.784,Z 341.401,A -85,B 0,C 180,E1 -5235.383,E2 -5235.383} C_VEL
LIN {X 0,Y 640.791,Z 341.407,A -85,B 0,C 180,E1 -5238.562,E2 -5238.562} C_VEL
LIN {X 0,Y 640.782,Z 341.405,A -85,B 0,C 180,E1 -5241.416,E2 -5241.416} C_VEL
LIN {X 0,Y 640.794,Z 341.406,A -85,B 0,C 180,E1 -5244.622,E2 -5244.622} C_VEL
LIN {X 0,Y 640.776,Z 341.402,A -85,B 0,C 180,E1 -5247.409,E2 -5247.409} C_VEL
LIN {X 0,Y 640.818,Z 341.403,A -85,B 0,C 180,E1 -5250.537,E2 -5250.537} C_VEL
LIN {X 0,Y 640.772,Z 341.408,A -85,B 0,C 180,E1 -5253.425,E2 -5253.425} C_VEL
LIN {X 0,Y 640.827,Z 341.407,A -85,B 0,C 180,E1 -5256.529,E2 -5256.529} C_VEL
LIN {X 0,Y 640.772,Z 341.409,A -85,B 0,C 180,E1 -5259.428,E2 -5259.428} C_VEL
LIN {X 0,Y 640.834,Z 341.405,A -85,B 0,C 180,E1 -5262.437,E2 -5262.437} C_VEL
LIN {X 0,Y 640.772,Z 341.409,A -85,B 0,C 180,E1 -5265.396,E2 -5265.396} C_VEL
LIN {X 0,Y 640.771,Z 341.41,A -85,B 0,C 180,E1 -5265.516,E2 -5265.516} C_VEL
LIN {X 0,Y 639.805,Z 341.536,A -85,B 0,C 180,E1 -5266.204,E2 -5266.204} C_VEL
LIN {X 0,Y 633.441,Z 342.33,A -85,B 0,C 180,E1 -5268.136,E2 -5268.136} C_VEL
LIN {X 0,Y 632.899,Z 342.393,A -85,B 0,C 180,E1 -5268.638,E2 -5268.638} C_VEL
LIN {X 0,Y 632.899,Z 342.475,A -85,B 0,C 180,E1 -5268.792,E2 -5268.792} C_VEL
LIN {X 0,Y 635.732,Z 349.946,A -85,B 0,C 180,E1 -5269.696,E2 -5269.696} C_VEL
LIN {X 0,Y 651.929,Z 376.386,A -85,B 0,C 180,E1 -5271.27,E2 -5271.27} C_VEL
LIN {X 0,Y 655.219,Z 382.606,A -85,B 0,C 180,E1 -5271.588,E2 -5271.588} C_VEL
LIN {X 0,Y 651.734,Z 625.825,A -85,B 0,C 180,E1 -5274.641,E2 -5274.641} C_VEL
LIN {X 0,Y 650.103,Z 738.43,A -85,B 0,C 180,E1 -5276.054,E2 -5276.054} C_VEL
LIN {X 0,Y 649.255,Z 763.755,A -85,B 0,C 180,E1 -5276.528,E2 -5276.528} C_VEL
LIN {X 0,Y 648.344,Z 784.02,A -85,B 0,C 180,E1 -5277.037,E2 -5277.037} C_VEL
LIN {X 0,Y 647.199,Z 806.535,A -85,B 0,C 180,E1 -5277.739,E2 -5277.739} C_VEL
LIN {X 0,Y 645.761,Z 828.658,A -85,B 0,C 180,E1 -5278.599,E2 -5278.599} C_VEL
LIN {X 0,Y 644.448,Z 848.584,A -85,B 0,C 180,E1 -5279.512,E2 -5279.512} C_VEL
LIN {X 0,Y 642.771,Z 871.115,A -85,B 0,C 180,E1 -5280.729,E2 -5280.729} C_VEL
LIN {X 0,Y 641.23,Z 890.778,A -85,B 0,C 180,E1 -5281.956,E2 -5281.956} C_VEL
LIN {X 0,Y 639.568,Z 912.054,A -85,B 0,C 180,E1 -5283.491,E2 -5283.491} C_VEL
LIN {X 0,Y 638.222,Z 929.12,A -85,B 0,C 180,E1 -5284.897,E2 -5284.897} C_VEL
LIN {X 0,Y 636.716,Z 948.611,A -85,B 0,C 180,E1 -5286.734,E2 -5286.734} C_VEL
LIN {X 0,Y 635.587,Z 964.079,A -85,B 0,C 180,E1 -5288.4,E2 -5288.4} C_VEL
LIN {X 0,Y 634.502,Z 980.189,A -85,B 0,C 180,E1 -5290.387,E2 -5290.387} C_VEL
LIN {X 0,Y 633.717,Z 992.853,A -85,B 0,C 180,E1 -5292.176,E2 -5292.176} C_VEL
LIN {X 0,Y 633.03,Z 1006.043,A -85,B 0,C 180,E1 -5294.33,E2 -5294.33} C_VEL
LIN {X 0,Y 632.607,Z 1015.8,A -85,B 0,C 180,E1 -5296.192,E2 -5296.192} C_VEL
LIN {X 0,Y 632.268,Z 1025.661,A -85,B 0,C 180,E1 -5298.414,E2 -5298.414} C_VEL
LIN {X 0,Y 632.076,Z 1032.667,A -85,B 0,C 180,E1 -5300.347,E2 -5300.347} C_VEL
LIN {X 0,Y 631.961,Z 1038.891,A -85,B 0,C 180,E1 -5302.454,E2 -5302.454} C_VEL
LIN {X 0,Y 631.918,Z 1043.416,A -85,B 0,C 180,E1 -5304.552,E2 -5304.552} C_VEL
LIN {X 0,Y 631.913,Z 1046.294,A -85,B 0,C 180,E1 -5306.462,E2 -5306.462} C_VEL
LIN {X 0,Y 631.904,Z 1048.18,A -85,B 0,C 180,E1 -5308.731,E2 -5308.731} C_VEL
LIN {X 0,Y 631.898,Z 1048.339,A -85,B 0,C 180,E1 -5310.725,E2 -5310.725} C_VEL
LIN {X 0,Y 631.899,Z 1047.326,A -85,B 0,C 180,E1 -5312.63,E2 -5312.63} C_VEL
LIN {X 0,Y 631.92,Z 1044.53,A -85,B 0,C 180,E1 -5314.902,E2 -5314.902} C_VEL
LIN {X 0,Y 631.946,Z 1040.791,A -85,B 0,C 180,E1 -5316.815,E2 -5316.815} C_VEL
LIN {X 0,Y 632.02,Z 1035.327,A -85,B 0,C 180,E1 -5318.919,E2 -5318.919} C_VEL
LIN {X 0,Y 632.185,Z 1028.129,A -85,B 0,C 180,E1 -5321.033,E2 -5321.033} C_VEL
LIN {X 0,Y 632.435,Z 1020.541,A -85,B 0,C 180,E1 -5322.881,E2 -5322.881} C_VEL
LIN {X 0,Y 632.881,Z 1009.501,A -85,B 0,C 180,E1 -5325.132,E2 -5325.132} C_VEL
LIN {X 0,Y 633.4,Z 998.813,A -85,B 0,C 180,E1 -5326.98,E2 -5326.98} C_VEL
LIN {X 0,Y 634.186,Z 985.049,A -85,B 0,C 180,E1 -5329.048,E2 -5329.048} C_VEL
LIN {X 0,Y 635.095,Z 971.206,A -85,B 0,C 180,E1 -5330.843,E2 -5330.843} C_VEL
LIN {X 0,Y 636.259,Z 954.909,A -85,B 0,C 180,E1 -5332.708,E2 -5332.708} C_VEL
LIN {X 0,Y 637.503,Z 938.271,A -85,B 0,C 180,E1 -5334.362,E2 -5334.362} C_VEL
LIN {X 0,Y 638.954,Z 919.839,A -85,B 0,C 180,E1 -5335.987,E2 -5335.987} C_VEL
LIN {X 0,Y 640.443,Z 900.993,A -85,B 0,C 180,E1 -5337.424,E2 -5337.424} C_VEL
LIN {X 0,Y 642.023,Z 881.079,A -85,B 0,C 180,E1 -5338.766,E2 -5338.766} C_VEL
LIN {X 0,Y 643.565,Z 860.343,A -85,B 0,C 180,E1 -5339.967,E2 -5339.967} C_VEL
LIN {X 0,Y 645.063,Z 839.843,A -85,B 0,C 180,E1 -5340.997,E2 -5340.997} C_VEL
LIN {X 0,Y 646.512,Z 817.703,A -85,B 0,C 180,E1 -5341.934,E2 -5341.934} C_VEL
LIN {X 0,Y 647.67,Z 797.289,A -85,B 0,C 180,E1 -5342.654,E2 -5342.654} C_VEL
LIN {X 0,Y 648.826,Z 774.038,A -85,B 0,C 180,E1 -5343.326,E2 -5343.326} C_VEL
LIN {X 0,Y 649.712,Z 750.566,A -85,B 0,C 180,E1 -5343.83,E2 -5343.83} C_VEL
LIN {X 0,Y 650.382,Z 726.055,A -85,B 0,C 180,E1 -5344.211,E2 -5344.211} C_VEL
LIN {X 0,Y 653.933,Z 471.494,A -85,B 0,C 180,E1 -5347.377,E2 -5347.377} C_VEL
LIN {X 0,Y 655.112,Z 382.017,A -85,B 0,C 180,E1 -5348.518,E2 -5348.518} C_VEL
LIN {X 0,Y 644.402,Z 363.92,A -85,B 0,C 180,E1 -5349.54,E2 -5349.54} C_VEL
LIN {X 0,Y 635.385,Z 349.19,A -85,B 0,C 180,E1 -5350.459,E2 -5350.459} C_VEL
LIN {X 0,Y 632.894,Z 342.392,A -85,B 0,C 180,E1 -5351.329,E2 -5351.329} C_VEL
LIN {X 0,Y 632.824,Z 342.375,A -85,B 0,C 180,E1 -5354.424,E2 -5354.424} C_VEL
LIN {X 0,Y 632.874,Z 342.381,A -85,B 0,C 180,E1 -5357.329,E2 -5357.329} C_VEL
LIN {X 0,Y 632.831,Z 342.396,A -85,B 0,C 180,E1 -5360.45,E2 -5360.45} C_VEL
LIN {X 0,Y 632.864,Z 342.393,A -85,B 0,C 180,E1 -5363.329,E2 -5363.329} C_VEL
LIN {X 0,Y 632.836,Z 342.396,A -85,B 0,C 180,E1 -5366.426,E2 -5366.426} C_VEL
LIN {X 0,Y 632.846,Z 342.392,A -85,B 0,C 180,E1 -5369.262,E2 -5369.262} C_VEL
LIN {X 0,Y 632.841,Z 342.388,A -85,B 0,C 180,E1 -5372.423,E2 -5372.423} C_VEL
LIN {X 0,Y 632.837,Z 342.401,A -85,B 0,C 180,E1 -5375.247,E2 -5375.247} C_VEL
LIN {X 0,Y 632.846,Z 342.396,A -85,B 0,C 180,E1 -5378.496,E2 -5378.496} C_VEL
LIN {X 0,Y 632.833,Z 342.392,A -85,B 0,C 180,E1 -5381.292,E2 -5381.292} C_VEL
LIN {X 0,Y 632.864,Z 342.384,A -85,B 0,C 180,E1 -5384.419,E2 -5384.419} C_VEL
LIN {X 0,Y 632.827,Z 342.399,A -85,B 0,C 180,E1 -5387.22,E2 -5387.22} C_VEL
LIN {X 0,Y 632.891,Z 342.394,A -85,B 0,C 180,E1 -5390.268,E2 -5390.268} C_VEL
LIN {X 0,Y 632.823,Z 342.392,A -85,B 0,C 180,E1 -5393.194,E2 -5393.194} C_VEL
LIN {X 0,Y 632.893,Z 342.397,A -85,B 0,C 180,E1 -5396.195,E2 -5396.195} C_VEL
LIN {X 0,Y 632.824,Z 342.391,A -85,B 0,C 180,E1 -5399.276,E2 -5399.276} C_VEL
LIN {X 0,Y 632.891,Z 342.386,A -85,B 0,C 180,E1 -5402.264,E2 -5402.264} C_VEL
LIN {X 0,Y 632.825,Z 342.398,A -85,B 0,C 180,E1 -5405.349,E2 -5405.349} C_VEL
LIN {X 0,Y 632.885,Z 342.387,A -85,B 0,C 180,E1 -5408.266,E2 -5408.266} C_VEL
LIN {X 0,Y 632.828,Z 342.393,A -85,B 0,C 180,E1 -5411.299,E2 -5411.299} C_VEL
LIN {X 0,Y 632.862,Z 342.398,A -85,B 0,C 180,E1 -5414.176,E2 -5414.176} C_VEL
LIN {X 0,Y 632.834,Z 342.392,A -85,B 0,C 180,E1 -5417.28,E2 -5417.28} C_VEL
LIN {X 0,Y 632.839,Z 342.397,A -85,B 0,C 180,E1 -5420.051,E2 -5420.051} C_VEL
LIN {X 0,Y 632.842,Z 342.394,A -85,B 0,C 180,E1 -5423.266,E2 -5423.266} C_VEL
LIN {X 0,Y 632.832,Z 342.398,A -85,B 0,C 180,E1 -5426.056,E2 -5426.056} C_VEL
LIN {X 0,Y 632.859,Z 342.397,A -85,B 0,C 180,E1 -5429.223,E2 -5429.223} C_VEL
LIN {X 0,Y 632.826,Z 342.396,A -85,B 0,C 180,E1 -5432.066,E2 -5432.066} C_VEL
LIN {X 0,Y 632.882,Z 342.397,A -85,B 0,C 180,E1 -5435.106,E2 -5435.106} C_VEL
LIN {X 0,Y 632.824,Z 342.4,A -85,B 0,C 180,E1 -5438.041,E2 -5438.041} C_VEL
LIN {X 0,Y 632.893,Z 342.366,A -85,B 0,C 180,E1 -5441.097,E2 -5441.097} C_VEL
LIN {X 0,Y 632.824,Z 342.397,A -85,B 0,C 180,E1 -5444.045,E2 -5444.045} C_VEL
LIN {X 0,Y 632.853,Z 342.47,A -85,B 0,C 180,E1 -5446.559,E2 -5446.559} C_VEL
LIN {X 0,Y 641.717,Z 365.187,A -85,B 0,C 180,E1 -5449.242,E2 -5449.242} C_VEL
LIN {X 0,Y 645.694,Z 375.698,A -85,B 0,C 180,E1 -5450.391,E2 -5450.391} C_VEL
LIN {X 0,Y 649.797,Z 383.306,A -85,B 0,C 180,E1 -5450.794,E2 -5450.794} C_VEL
LIN {X 0,Y 655.155,Z 406.534,A -85,B 0,C 180,E1 -5451.491,E2 -5451.491} C_VEL
LIN {X 0,Y 651.368,Z 674.653,A -85,B 0,C 180,E1 -5454.843,E2 -5454.843} C_VEL
LIN {X 0,Y 650.018,Z 767.47,A -85,B 0,C 180,E1 -5456.009,E2 -5456.009} C_VEL
LIN {X 0,Y 649.156,Z 792.846,A -85,B 0,C 180,E1 -5456.482,E2 -5456.482} C_VEL
LIN {X 0,Y 648.244,Z 813.081,A -85,B 0,C 180,E1 -5456.987,E2 -5456.987} C_VEL
LIN {X 0,Y 647.095,Z 835.951,A -85,B 0,C 180,E1 -5457.696,E2 -5457.696} C_VEL
LIN {X 0,Y 645.645,Z 858.663,A -85,B 0,C 180,E1 -5458.575,E2 -5458.575} C_VEL
LIN {X 0,Y 644.282,Z 880.098,A -85,B 0,C 180,E1 -5459.555,E2 -5459.555} C_VEL
LIN {X 0,Y 642.66,Z 902.269,A -85,B 0,C 180,E1 -5460.755,E2 -5460.755} C_VEL
LIN {X 0,Y 641.294,Z 919.981,A -85,B 0,C 180,E1 -5461.858,E2 -5461.858} C_VEL
LIN {X 0,Y 639.606,Z 941.567,A -85,B 0,C 180,E1 -5463.407,E2 -5463.407} C_VEL
LIN {X 0,Y 638.282,Z 958.284,A -85,B 0,C 180,E1 -5464.78,E2 -5464.78} C_VEL
LIN {X 0,Y 636.866,Z 976.748,A -85,B 0,C 180,E1 -5466.498,E2 -5466.498} C_VEL
LIN {X 0,Y 635.733,Z 991.985,A -85,B 0,C 180,E1 -5468.12,E2 -5468.12} C_VEL
LIN {X 0,Y 634.665,Z 1007.703,A -85,B 0,C 180,E1 -5470.009,E2 -5470.009} C_VEL
LIN {X 0,Y 633.812,Z 1021.245,A -85,B 0,C 180,E1 -5471.893,E2 -5471.893} C_VEL
LIN {X 0,Y 633.141,Z 1034.211,A -85,B 0,C 180,E1 -5473.956,E2 -5473.956} C_VEL
LIN {X 0,Y 632.654,Z 1044.642,A -85,B 0,C 180,E1 -5475.913,E2 -5475.913} C_VEL
LIN {X 0,Y 632.316,Z 1053.991,A -85,B 0,C 180,E1 -5477.952,E2 -5477.952} C_VEL
LIN {X 0,Y 632.086,Z 1061.907,A -85,B 0,C 180,E1 -5480.071,E2 -5480.071} C_VEL
LIN {X 0,Y 631.983,Z 1067.744,A -85,B 0,C 180,E1 -5481.997,E2 -5481.997} C_VEL
LIN {X 0,Y 631.933,Z 1073.016,A -85,B 0,C 180,E1 -5484.279,E2 -5484.279} C_VEL
LIN {X 0,Y 631.906,Z 1076.124,A -85,B 0,C 180,E1 -5486.28,E2 -5486.28} C_VEL
LIN {X 0,Y 631.896,Z 1077.969,A -85,B 0,C 180,E1 -5488.277,E2 -5488.277} C_VEL
LIN {X 0,Y 631.893,Z 1078.395,A -85,B 0,C 180,E1 -5490.453,E2 -5490.453} C_VEL
LIN {X 0,Y 631.909,Z 1077.428,A -85,B 0,C 180,E1 -5492.449,E2 -5492.449} C_VEL
LIN {X 0,Y 631.922,Z 1074.768,A -85,B 0,C 180,E1 -5494.72,E2 -5494.72} C_VEL
LIN {X 0,Y 631.937,Z 1070.896,A -85,B 0,C 180,E1 -5496.724,E2 -5496.724} C_VEL
LIN {X 0,Y 632.01,Z 1065.711,A -85,B 0,C 180,E1 -5498.736,E2 -5498.736} C_VEL
LIN {X 0,Y 632.187,Z 1058.309,A -85,B 0,C 180,E1 -5500.941,E2 -5500.941} C_VEL
LIN {X 0,Y 632.439,Z 1050.346,A -85,B 0,C 180,E1 -5502.881,E2 -5502.881} C_VEL
LIN {X 0,Y 632.886,Z 1039.248,A -85,B 0,C 180,E1 -5505.134,E2 -5505.134} C_VEL
LIN {X 0,Y 633.408,Z 1028.545,A -85,B 0,C 180,E1 -5506.98,E2 -5506.98} C_VEL
LIN {X 0,Y 634.203,Z 1014.722,A -85,B 0,C 180,E1 -5509.048,E2 -5509.048} C_VEL
LIN {X 0,Y 635.123,Z 1000.848,A -85,B 0,C 180,E1 -5510.842,E2 -5510.842} C_VEL
LIN {X 0,Y 636.307,Z 984.156,A -85,B 0,C 180,E1 -5512.741,E2 -5512.741} C_VEL
LIN {X 0,Y 637.505,Z 968.256,A -85,B 0,C 180,E1 -5514.319,E2 -5514.319} C_VEL
LIN {X 0,Y 638.959,Z 949.759,A -85,B 0,C 180,E1 -5515.948,E2 -5515.948} C_VEL
LIN {X 0,Y 640.431,Z 931.06,A -85,B 0,C 180,E1 -5517.374,E2 -5517.374} C_VEL
LIN {X 0,Y 642.047,Z 910.746,A -85,B 0,C 180,E1 -5518.742,E2 -5518.742} C_VEL
LIN {X 0,Y 643.519,Z 890.232,A -85,B 0,C 180,E1 -5519.918,E2 -5519.918} C_VEL
LIN {X 0,Y 644.949,Z 870,A -85,B 0,C 180,E1 -5520.926,E2 -5520.926} C_VEL
LIN {X 0,Y 646.408,Z 847.181,A -85,B 0,C 180,E1 -5521.887,E2 -5521.887} C_VEL
LIN {X 0,Y 647.553,Z 826.627,A -85,B 0,C 180,E1 -5522.608,E2 -5522.608} C_VEL
LIN {X 0,Y 648.717,Z 803.17,A -85,B 0,C 180,E1 -5523.282,E2 -5523.282} C_VEL
LIN {X 0,Y 649.635,Z 779.421,A -85,B 0,C 180,E1 -5523.789,E2 -5523.789} C_VEL
LIN {X 0,Y 650.31,Z 754.896,A -85,B 0,C 180,E1 -5524.169,E2 -5524.169} C_VEL
LIN {X 0,Y 653.691,Z 505.872,A -85,B 0,C 180,E1 -5527.258,E2 -5527.258} C_VEL
LIN {X 0,Y 654.988,Z 404.941,A -85,B 0,C 180,E1 -5528.542,E2 -5528.542} C_VEL
LIN {X 0,Y 649.27,Z 381.895,A -85,B 0,C 180,E1 -5529.264,E2 -5529.264} C_VEL
LIN {X 0,Y 645.391,Z 374.974,A -85,B 0,C 180,E1 -5529.665,E2 -5529.665} C_VEL
LIN {X 0,Y 637.865,Z 355.358,A -85,B 0,C 180,E1 -5531.896,E2 -5531.896} C_VEL
LIN {X 0,Y 633.522,Z 344.707,A -85,B 0,C 180,E1 -5533.182,E2 -5533.182} C_VEL
LIN {X 0,Y 632.843,Z 342.398,A -85,B 0,C 180,E1 -5533.473,E2 -5533.473} C_VEL
LIN {X 0,Y 632.833,Z 342.399,A -85,B 0,C 180,E1 -5536.225,E2 -5536.225} C_VEL
LIN {X 0,Y 632.863,Z 342.398,A -85,B 0,C 180,E1 -5539.387,E2 -5539.387} C_VEL
LIN {X 0,Y 632.827,Z 342.397,A -85,B 0,C 180,E1 -5542.189,E2 -5542.189} C_VEL
LIN {X 0,Y 632.885,Z 342.361,A -85,B 0,C 180,E1 -5545.239,E2 -5545.239} C_VEL
LIN {X 0,Y 632.823,Z 342.393,A -85,B 0,C 180,E1 -5548.147,E2 -5548.147} C_VEL
LIN {X 0,Y 632.897,Z 342.394,A -85,B 0,C 180,E1 -5551.09,E2 -5551.09} C_VEL
LIN {X 0,Y 632.828,Z 342.399,A -85,B 0,C 180,E1 -5554.145,E2 -5554.145} C_VEL
LIN {X 0,Y 632.89,Z 342.389,A -85,B 0,C 180,E1 -5557.129,E2 -5557.129} C_VEL
LIN {X 0,Y 632.83,Z 342.395,A -85,B 0,C 180,E1 -5560.141,E2 -5560.141} C_VEL
LIN {X 0,Y 632.862,Z 342.394,A -85,B 0,C 180,E1 -5563.005,E2 -5563.005} C_VEL
LIN {X 0,Y 632.841,Z 342.399,A -85,B 0,C 180,E1 -5566.104,E2 -5566.104} C_VEL
LIN {X 0,Y 632.848,Z 342.387,A -85,B 0,C 180,E1 -5568.978,E2 -5568.978} C_VEL
LIN {X 0,Y 632.841,Z 342.386,A -85,B 0,C 180,E1 -5572.19,E2 -5572.19} C_VEL
LIN {X 0,Y 632.843,Z 342.396,A -85,B 0,C 180,E1 -5575.015,E2 -5575.015} C_VEL
LIN {X 0,Y 632.844,Z 342.398,A -85,B 0,C 180,E1 -5578.28,E2 -5578.28} C_VEL
LIN {X 0,Y 632.841,Z 342.393,A -85,B 0,C 180,E1 -5581.086,E2 -5581.086} C_VEL
LIN {X 0,Y 632.847,Z 342.4,A -85,B 0,C 180,E1 -5584.349,E2 -5584.349} C_VEL
LIN {X 0,Y 632.839,Z 342.385,A -85,B 0,C 180,E1 -5587.17,E2 -5587.17} C_VEL
LIN {X 0,Y 632.853,Z 342.39,A -85,B 0,C 180,E1 -5590.377,E2 -5590.377} C_VEL
LIN {X 0,Y 632.841,Z 342.396,A -85,B 0,C 180,E1 -5593.275,E2 -5593.275} C_VEL
LIN {X 0,Y 632.851,Z 342.395,A -85,B 0,C 180,E1 -5596.523,E2 -5596.523} C_VEL
LIN {X 0,Y 632.844,Z 342.392,A -85,B 0,C 180,E1 -5599.394,E2 -5599.394} C_VEL
LIN {X 0,Y 632.849,Z 342.396,A -85,B 0,C 180,E1 -5602.676,E2 -5602.676} C_VEL
LIN {X 0,Y 632.848,Z 342.395,A -85,B 0,C 180,E1 -5605.555,E2 -5605.555} C_VEL
LIN {X 0,Y 632.848,Z 342.401,A -85,B 0,C 180,E1 -5608.809,E2 -5608.809} C_VEL
LIN {X 0,Y 632.846,Z 342.387,A -85,B 0,C 180,E1 -5611.639,E2 -5611.639} C_VEL
LIN {X 0,Y 632.847,Z 342.395,A -85,B 0,C 180,E1 -5614.914,E2 -5614.914} C_VEL
LIN {X 0,Y 632.852,Z 342.388,A -85,B 0,C 180,E1 -5617.816,E2 -5617.816} C_VEL
LIN {X 0,Y 632.85,Z 342.399,A -85,B 0,C 180,E1 -5620.972,E2 -5620.972} C_VEL
LIN {X 0,Y 632.845,Z 342.4,A -85,B 0,C 180,E1 -5623.792,E2 -5623.792} C_VEL
LIN {X 0,Y 632.85,Z 342.396,A -85,B 0,C 180,E1 -5627.081,E2 -5627.081} C_VEL
LIN {X 0,Y 632.899,Z 342.393,A -85,B 0,C 180,E1 -5628.638,E2 -5628.638} C_VEL
LIN {X 0,Y 633.627,Z 343.05,A -85,B 0,C 180,E1 -5628.896,E2 -5628.896} C_VEL
LIN {X 0,Y 634.487,Z 345.317,A -85,B 0,C 180,E1 -5629.194,E2 -5629.194} C_VEL
LIN {X 0,Y 634.821,Z 349.511,A -85,B 0,C 180,E1 -5629.515,E2 -5629.515} C_VEL
LIN {X 0,Y 635.335,Z 353.938,A -85,B 0,C 180,E1 -5629.724,E2 -5629.724} C_VEL
LIN {X 0,Y 638.798,Z 367.048,A -85,B 0,C 180,E1 -5630.175,E2 -5630.175} C_VEL
LIN {X 0,Y 640.604,Z 371.149,A -85,B 0,C 180,E1 -5630.371,E2 -5630.371} C_VEL
LIN {X 0,Y 648.926,Z 385.362,A -85,B 0,C 180,E1 -5631.181,E2 -5631.181} C_VEL
LIN {X 0,Y 645.176,Z 629.429,A -85,B 0,C 180,E1 -5634.271,E2 -5634.271} C_VEL
LIN {X 0,Y 643.478,Z 738.686,A -85,B 0,C 180,E1 -5635.656,E2 -5635.656} C_VEL
LIN {X 0,Y 642.583,Z 763.996,A -85,B 0,C 180,E1 -5636.134,E2 -5636.134} C_VEL
LIN {X 0,Y 641.629,Z 784.081,A -85,B 0,C 180,E1 -5636.641,E2 -5636.641} C_VEL
LIN {X 0,Y 640.445,Z 806.049,A -85,B 0,C 180,E1 -5637.33,E2 -5637.33} C_VEL
LIN {X 0,Y 638.872,Z 828.887,A -85,B 0,C 180,E1 -5638.221,E2 -5638.221} C_VEL
LIN {X 0,Y 637.403,Z 849.812,A -85,B 0,C 180,E1 -5639.191,E2 -5639.191} C_VEL
LIN {X 0,Y 635.638,Z 871.851,A -85,B 0,C 180,E1 -5640.4,E2 -5640.4} C_VEL
LIN {X 0,Y 634.085,Z 890.194,A -85,B 0,C 180,E1 -5641.561,E2 -5641.561} C_VEL
LIN {X 0,Y 632.239,Z 911.623,A -85,B 0,C 180,E1 -5643.122,E2 -5643.122} C_VEL
LIN {X 0,Y 630.81,Z 928.577,A -85,B 0,C 180,E1 -5644.531,E2 -5644.531} C_VEL
LIN {X 0,Y 629.248,Z 947.256,A -85,B 0,C 180,E1 -5646.295,E2 -5646.295} C_VEL
LIN {X 0,Y 628.049,Z 962.393,A -85,B 0,C 180,E1 -5647.931,E2 -5647.931} C_VEL
LIN {X 0,Y 626.885,Z 978.086,A -85,B 0,C 180,E1 -5649.847,E2 -5649.847} C_VEL
LIN {X 0,Y 625.969,Z 991.585,A -85,B 0,C 180,E1 -5651.755,E2 -5651.755} C_VEL
LIN {X 0,Y 625.236,Z 1004.492,A -85,B 0,C 180,E1 -5653.843,E2 -5653.843} C_VEL
LIN {X 0,Y 624.715,Z 1014.885,A -85,B 0,C 180,E1 -5655.825,E2 -5655.825} C_VEL
LIN {X 0,Y 624.344,Z 1024.595,A -85,B 0,C 180,E1 -5657.983,E2 -5657.983} C_VEL
LIN {X 0,Y 624.095,Z 1032.366,A -85,B 0,C 180,E1 -5660.129,E2 -5660.129} C_VEL
LIN {X 0,Y 623.984,Z 1038.13,A -85,B 0,C 180,E1 -5662.079,E2 -5662.079} C_VEL
LIN {X 0,Y 623.924,Z 1043.257,A -85,B 0,C 180,E1 -5664.39,E2 -5664.39} C_VEL
LIN {X 0,Y 623.913,Z 1046.181,A -85,B 0,C 180,E1 -5666.325,E2 -5666.325} C_VEL
LIN {X 0,Y 623.896,Z 1048.13,A -85,B 0,C 180,E1 -5668.531,E2 -5668.531} C_VEL
LIN {X 0,Y 623.895,Z 1048.361,A -85,B 0,C 180,E1 -5670.643,E2 -5670.643} C_VEL
LIN {X 0,Y 623.902,Z 1047.394,A -85,B 0,C 180,E1 -5672.572,E2 -5672.572} C_VEL
LIN {X 0,Y 623.921,Z 1044.688,A -85,B 0,C 180,E1 -5674.872,E2 -5674.872} C_VEL
LIN {X 0,Y 623.955,Z 1040.79,A -85,B 0,C 180,E1 -5676.903,E2 -5676.903} C_VEL
LIN {X 0,Y 624.035,Z 1035.325,A -85,B 0,C 180,E1 -5679.034,E2 -5679.034} C_VEL
LIN {X 0,Y 624.214,Z 1028.126,A -85,B 0,C 180,E1 -5681.176,E2 -5681.176} C_VEL
LIN {X 0,Y 624.484,Z 1020.537,A -85,B 0,C 180,E1 -5683.048,E2 -5683.048} C_VEL
LIN {X 0,Y 624.966,Z 1009.615,A -85,B 0,C 180,E1 -5685.307,E2 -5685.307} C_VEL
LIN {X 0,Y 625.545,Z 998.808,A -85,B 0,C 180,E1 -5687.2,E2 -5687.2} C_VEL
LIN {X 0,Y 626.396,Z 985.043,A -85,B 0,C 180,E1 -5689.295,E2 -5689.295} C_VEL
LIN {X 0,Y 627.38,Z 971.199,A -85,B 0,C 180,E1 -5691.112,E2 -5691.112} C_VEL
LIN {X 0,Y 628.602,Z 955.5,A -85,B 0,C 180,E1 -5692.937,E2 -5692.937} C_VEL
LIN {X 0,Y 629.947,Z 938.771,A -85,B 0,C 180,E1 -5694.624,E2 -5694.624} C_VEL
LIN {X 0,Y 631.508,Z 920.434,A -85,B 0,C 180,E1 -5696.266,E2 -5696.266} C_VEL
LIN {X 0,Y 633.159,Z 901.028,A -85,B 0,C 180,E1 -5697.766,E2 -5697.766} C_VEL
LIN {X 0,Y 634.872,Z 881.265,A -85,B 0,C 180,E1 -5699.121,E2 -5699.121} C_VEL
LIN {X 0,Y 636.538,Z 860.548,A -85,B 0,C 180,E1 -5700.333,E2 -5700.333} C_VEL
LIN {X 0,Y 638.09,Z 840.529,A -85,B 0,C 180,E1 -5701.349,E2 -5701.349} C_VEL
LIN {X 0,Y 639.672,Z 817.902,A -85,B 0,C 180,E1 -5702.316,E2 -5702.316} C_VEL
LIN {X 0,Y 640.9,Z 797.485,A -85,B 0,C 180,E1 -5703.043,E2 -5703.043} C_VEL
LIN {X 0,Y 642.133,Z 774.064,A -85,B 0,C 180,E1 -5703.723,E2 -5703.723} C_VEL
LIN {X 0,Y 643.079,Z 750.607,A -85,B 0,C 180,E1 -5704.23,E2 -5704.23} C_VEL
LIN {X 0,Y 643.779,Z 726.037,A -85,B 0,C 180,E1 -5704.614,E2 -5704.614} C_VEL
LIN {X 0,Y 647.583,Z 471.784,A -85,B 0,C 180,E1 -5707.805,E2 -5707.805} C_VEL
LIN {X 0,Y 648.753,Z 385.021,A -85,B 0,C 180,E1 -5708.927,E2 -5708.927} C_VEL
LIN {X 0,Y 635.412,Z 362.646,A -85,B 0,C 180,E1 -5710.235,E2 -5710.235} C_VEL
LIN {X 0,Y 627.271,Z 349.775,A -85,B 0,C 180,E1 -5711.064,E2 -5711.064} C_VEL
LIN {X 0,Y 624.926,Z 343.391,A -85,B 0,C 180,E1 -5711.884,E2 -5711.884} C_VEL
LIN {X 0,Y 624.888,Z 343.366,A -85,B 0,C 180,E1 -5714.753,E2 -5714.753} C_VEL
LIN {X 0,Y 624.943,Z 343.357,A -85,B 0,C 180,E1 -5717.798,E2 -5717.798} C_VEL
LIN {X 0,Y 624.888,Z 343.387,A -85,B 0,C 180,E1 -5720.756,E2 -5720.756} C_VEL
LIN {X 0,Y 624.953,Z 343.387,A -85,B 0,C 180,E1 -5723.816,E2 -5723.816} C_VEL
LIN {X 0,Y 624.887,Z 343.387,A -85,B 0,C 180,E1 -5726.822,E2 -5726.822} C_VEL
LIN {X 0,Y 624.961,Z 343.381,A -85,B 0,C 180,E1 -5729.842,E2 -5729.842} C_VEL
LIN {X 0,Y 624.886,Z 343.378,A -85,B 0,C 180,E1 -5732.868,E2 -5732.868} C_VEL
LIN {X 0,Y 624.956,Z 343.374,A -85,B 0,C 180,E1 -5735.922,E2 -5735.922} C_VEL
LIN {X 0,Y 624.888,Z 343.387,A -85,B 0,C 180,E1 -5738.898,E2 -5738.898} C_VEL
LIN {X 0,Y 624.952,Z 343.385,A -85,B 0,C 180,E1 -5741.917,E2 -5741.917} C_VEL
LIN {X 0,Y 624.885,Z 343.376,A -85,B 0,C 180,E1 -5744.976,E2 -5744.976} C_VEL
LIN {X 0,Y 624.941,Z 343.381,A -85,B 0,C 180,E1 -5747.901,E2 -5747.901} C_VEL
LIN {X 0,Y 624.889,Z 343.386,A -85,B 0,C 180,E1 -5750.978,E2 -5750.978} C_VEL
LIN {X 0,Y 624.923,Z 343.376,A -85,B 0,C 180,E1 -5753.846,E2 -5753.846} C_VEL
LIN {X 0,Y 624.894,Z 343.384,A -85,B 0,C 180,E1 -5756.973,E2 -5756.973} C_VEL
LIN {X 0,Y 624.909,Z 343.382,A -85,B 0,C 180,E1 -5759.817,E2 -5759.817} C_VEL
LIN {X 0,Y 624.896,Z 343.371,A -85,B 0,C 180,E1 -5763.027,E2 -5763.027} C_VEL
LIN {X 0,Y 624.906,Z 343.39,A -85,B 0,C 180,E1 -5765.878,E2 -5765.878} C_VEL
LIN {X 0,Y 624.898,Z 343.385,A -85,B 0,C 180,E1 -5769.115,E2 -5769.115} C_VEL
LIN {X 0,Y 624.908,Z 343.38,A -85,B 0,C 180,E1 -5772.006,E2 -5772.006} C_VEL
LIN {X 0,Y 624.896,Z 343.384,A -85,B 0,C 180,E1 -5775.235,E2 -5775.235} C_VEL
LIN {X 0,Y 624.904,Z 343.384,A -85,B 0,C 180,E1 -5778.084,E2 -5778.084} C_VEL
LIN {X 0,Y 624.9,Z 343.381,A -85,B 0,C 180,E1 -5781.298,E2 -5781.298} C_VEL
LIN {X 0,Y 624.898,Z 343.384,A -85,B 0,C 180,E1 -5784.081,E2 -5784.081} C_VEL
LIN {X 0,Y 624.901,Z 343.381,A -85,B 0,C 180,E1 -5787.372,E2 -5787.372} C_VEL
LIN {X 0,Y 624.898,Z 343.391,A -85,B 0,C 180,E1 -5790.161,E2 -5790.161} C_VEL
LIN {X 0,Y 624.907,Z 343.385,A -85,B 0,C 180,E1 -5793.396,E2 -5793.396} C_VEL
LIN {X 0,Y 624.895,Z 343.392,A -85,B 0,C 180,E1 -5796.25,E2 -5796.25} C_VEL
LIN {X 0,Y 624.913,Z 343.377,A -85,B 0,C 180,E1 -5799.436,E2 -5799.436} C_VEL
LIN {X 0,Y 624.888,Z 343.381,A -85,B 0,C 180,E1 -5802.225,E2 -5802.225} C_VEL
LIN {X 0,Y 624.932,Z 343.385,A -85,B 0,C 180,E1 -5805.38,E2 -5805.38} C_VEL
LIN {X 0,Y 624.913,Z 343.57,A -85,B 0,C 180,E1 -5805.992,E2 -5805.992} C_VEL
LIN {X 0,Y 633.695,Z 365.712,A -85,B 0,C 180,E1 -5808.683,E2 -5808.683} C_VEL
LIN {X 0,Y 637.444,Z 375.503,A -85,B 0,C 180,E1 -5809.775,E2 -5809.775} C_VEL
LIN {X 0,Y 644.065,Z 387.268,A -85,B 0,C 180,E1 -5810.435,E2 -5810.435} C_VEL
LIN {X 0,Y 648.852,Z 408.314,A -85,B 0,C 180,E1 -5811.074,E2 -5811.074} C_VEL
LIN {X 0,Y 644.797,Z 675.829,A -85,B 0,C 180,E1 -5814.449,E2 -5814.449} C_VEL
LIN {X 0,Y 643.362,Z 767.492,A -85,B 0,C 180,E1 -5815.612,E2 -5815.612} C_VEL
LIN {X 0,Y 642.444,Z 792.76,A -85,B 0,C 180,E1 -5816.088,E2 -5816.088} C_VEL
LIN {X 0,Y 641.477,Z 812.865,A -85,B 0,C 180,E1 -5816.594,E2 -5816.594} C_VEL
LIN {X 0,Y 640.276,Z 835.314,A -85,B 0,C 180,E1 -5817.294,E2 -5817.294} C_VEL
LIN {X 0,Y 638.714,Z 858.19,A -85,B 0,C 180,E1 -5818.182,E2 -5818.182} C_VEL
LIN {X 0,Y 637.226,Z 879.879,A -85,B 0,C 180,E1 -5819.181,E2 -5819.181} C_VEL
LIN {X 0,Y 635.566,Z 901.232,A -85,B 0,C 180,E1 -5820.345,E2 -5820.345} C_VEL
LIN {X 0,Y 634.055,Z 919.858,A -85,B 0,C 180,E1 -5821.508,E2 -5821.508} C_VEL
LIN {X 0,Y 632.281,Z 941.138,A -85,B 0,C 180,E1 -5823.038,E2 -5823.038} C_VEL
LIN {X 0,Y 630.831,Z 958.282,A -85,B 0,C 180,E1 -5824.461,E2 -5824.461} C_VEL
LIN {X 0,Y 629.293,Z 976.747,A -85,B 0,C 180,E1 -5826.198,E2 -5826.198} C_VEL
LIN {X 0,Y 628.078,Z 991.933,A -85,B 0,C 180,E1 -5827.833,E2 -5827.833} C_VEL
LIN {X 0,Y 626.91,Z 1007.705,A -85,B 0,C 180,E1 -5829.751,E2 -5829.751} C_VEL
LIN {X 0,Y 625.997,Z 1021.243,A -85,B 0,C 180,E1 -5831.659,E2 -5831.659} C_VEL
LIN {X 0,Y 625.286,Z 1033.689,A -85,B 0,C 180,E1 -5833.654,E2 -5833.654} C_VEL
LIN {X 0,Y 624.723,Z 1044.641,A -85,B 0,C 180,E1 -5835.73,E2 -5835.73} C_VEL
LIN {X 0,Y 624.367,Z 1053.585,A -85,B 0,C 180,E1 -5837.702,E2 -5837.702} C_VEL
LIN {X 0,Y 624.106,Z 1061.907,A -85,B 0,C 180,E1 -5839.943,E2 -5839.943} C_VEL
LIN {X 0,Y 624.01,Z 1067.49,A -85,B 0,C 180,E1 -5841.801,E2 -5841.801} C_VEL
LIN {X 0,Y 623.94,Z 1072.696,A -85,B 0,C 180,E1 -5844.021,E2 -5844.021} C_VEL
LIN {X 0,Y 623.907,Z 1076.01,A -85,B 0,C 180,E1 -5846.14,E2 -5846.14} C_VEL
LIN {X 0,Y 623.904,Z 1077.835,A -85,B 0,C 180,E1 -5848.071,E2 -5848.071} C_VEL
LIN {X 0,Y 623.895,Z 1078.417,A -85,B 0,C 180,E1 -5850.367,E2 -5850.367} C_VEL
LIN {X 0,Y 623.91,Z 1077.496,A -85,B 0,C 180,E1 -5852.388,E2 -5852.388} C_VEL
LIN {X 0,Y 623.919,Z 1075.085,A -85,B 0,C 180,E1 -5854.596,E2 -5854.596} C_VEL
LIN {X 0,Y 623.939,Z 1071.102,A -85,B 0,C 180,E1 -5856.718,E2 -5856.718} C_VEL
LIN {X 0,Y 624.014,Z 1066.219,A -85,B 0,C 180,E1 -5858.663,E2 -5858.663} C_VEL
LIN {X 0,Y 624.206,Z 1058.661,A -85,B 0,C 180,E1 -5860.989,E2 -5860.989} C_VEL
LIN {X 0,Y 624.476,Z 1050.75,A -85,B 0,C 180,E1 -5862.954,E2 -5862.954} C_VEL
LIN {X 0,Y 624.93,Z 1040.405,A -85,B 0,C 180,E1 -5865.117,E2 -5865.117} C_VEL
LIN {X 0,Y 625.518,Z 1029.117,A -85,B 0,C 180,E1 -5867.105,E2 -5867.105} C_VEL
LIN {X 0,Y 626.334,Z 1016.121,A -85,B 0,C 180,E1 -5869.103,E2 -5869.103} C_VEL
LIN {X 0,Y 627.355,Z 1001.616,A -85,B 0,C 180,E1 -5871.015,E2 -5871.015} C_VEL
LIN {X 0,Y 628.562,Z 986,A -85,B 0,C 180,E1 -5872.839,E2 -5872.839} C_VEL
LIN {X 0,Y 629.943,Z 968.824,A -85,B 0,C 180,E1 -5874.574,E2 -5874.574} C_VEL
LIN {X 0,Y 631.502,Z 950.499,A -85,B 0,C 180,E1 -5876.216,E2 -5876.216} C_VEL
LIN {X 0,Y 633.078,Z 931.695,A -85,B 0,C 180,E1 -5877.668,E2 -5877.668} C_VEL
LIN {X 0,Y 634.609,Z 913.191,A -85,B 0,C 180,E1 -5878.928,E2 -5878.928} C_VEL
LIN {X 0,Y 636.353,Z 890.919,A -85,B 0,C 180,E1 -5880.238,E2 -5880.238} C_VEL
LIN {X 0,Y 637.792,Z 871.803,A -85,B 0,C 180,E1 -5881.207,E2 -5881.207} C_VEL
LIN {X 0,Y 639.438,Z 848.237,A -85,B 0,C 180,E1 -5882.224,E2 -5882.224} C_VEL
LIN {X 0,Y 640.692,Z 827.154,A -85,B 0,C 180,E1 -5882.975,E2 -5882.975} C_VEL
LIN {X 0,Y 641.943,Z 803.834,A -85,B 0,C 180,E1 -5883.656,E2 -5883.656} C_VEL
LIN {X 0,Y 642.946,Z 779.736,A -85,B 0,C 180,E1 -5884.178,E2 -5884.178} C_VEL
LIN {X 0,Y 643.644,Z 756.117,A -85,B 0,C 180,E1 -5884.55,E2 -5884.55} C_VEL
LIN {X 0,Y 647.272,Z 508.08,A -85,B 0,C 180,E1 -5887.659,E2 -5887.659} C_VEL
LIN {X 0,Y 648.705,Z 406.814,A -85,B 0,C 180,E1 -5888.957,E2 -5888.957} C_VEL
LIN {X 0,Y 643.623,Z 386.088,A -85,B 0,C 180,E1 -5889.613,E2 -5889.613} C_VEL
LIN {X 0,Y 637.057,Z 374.684,A -85,B 0,C 180,E1 -5890.29,E2 -5890.29} C_VEL
LIN {X 0,Y 630.315,Z 357.127,A -85,B 0,C 180,E1 -5892.334,E2 -5892.334} C_VEL
LIN {X 0,Y 625.585,Z 345.795,A -85,B 0,C 180,E1 -5893.743,E2 -5893.743} C_VEL
LIN {X 0,Y 624.888,Z 343.388,A -85,B 0,C 180,E1 -5894.04,E2 -5894.04} C_VEL
LIN {X 0,Y 624.944,Z 343.386,A -85,B 0,C 180,E1 -5897.157,E2 -5897.157} C_VEL
LIN {X 0,Y 624.886,Z 343.383,A -85,B 0,C 180,E1 -5900.085,E2 -5900.085} C_VEL
LIN {X 0,Y 624.952,Z 343.355,A -85,B 0,C 180,E1 -5903.131,E2 -5903.131} C_VEL
LIN {X 0,Y 624.887,Z 343.381,A -85,B 0,C 180,E1 -5906.162,E2 -5906.162} C_VEL
LIN {X 0,Y 624.959,Z 343.373,A -85,B 0,C 180,E1 -5909.222,E2 -5909.222} C_VEL
LIN {X 0,Y 624.888,Z 343.376,A -85,B 0,C 180,E1 -5912.249,E2 -5912.249} C_VEL
LIN {X 0,Y 624.956,Z 343.377,A -85,B 0,C 180,E1 -5915.335,E2 -5915.335} C_VEL
LIN {X 0,Y 624.889,Z 343.387,A -85,B 0,C 180,E1 -5918.307,E2 -5918.307} C_VEL
LIN {X 0,Y 624.955,Z 343.381,A -85,B 0,C 180,E1 -5921.338,E2 -5921.338} C_VEL
LIN {X 0,Y 624.887,Z 343.381,A -85,B 0,C 180,E1 -5924.422,E2 -5924.422} C_VEL
LIN {X 0,Y 624.955,Z 343.379,A -85,B 0,C 180,E1 -5927.432,E2 -5927.432} C_VEL
LIN {X 0,Y 624.888,Z 343.388,A -85,B 0,C 180,E1 -5930.514,E2 -5930.514} C_VEL
LIN {X 0,Y 624.957,Z 343.371,A -85,B 0,C 180,E1 -5933.57,E2 -5933.57} C_VEL
LIN {X 0,Y 624.888,Z 343.379,A -85,B 0,C 180,E1 -5936.606,E2 -5936.606} C_VEL
LIN {X 0,Y 624.959,Z 343.383,A -85,B 0,C 180,E1 -5939.633,E2 -5939.633} C_VEL
LIN {X 0,Y 624.889,Z 343.382,A -85,B 0,C 180,E1 -5942.66,E2 -5942.66} C_VEL
LIN {X 0,Y 624.954,Z 343.382,A -85,B 0,C 180,E1 -5945.693,E2 -5945.693} C_VEL
LIN {X 0,Y 624.892,Z 343.388,A -85,B 0,C 180,E1 -5948.743,E2 -5948.743} C_VEL
LIN {X 0,Y 624.945,Z 343.371,A -85,B 0,C 180,E1 -5951.724,E2 -5951.724} C_VEL
LIN {X 0,Y 624.893,Z 343.381,A -85,B 0,C 180,E1 -5954.834,E2 -5954.834} C_VEL
LIN {X 0,Y 624.951,Z 343.382,A -85,B 0,C 180,E1 -5957.83,E2 -5957.83} C_VEL
LIN {X 0,Y 624.896,Z 343.386,A -85,B 0,C 180,E1 -5960.905,E2 -5960.905} C_VEL
LIN {X 0,Y 624.946,Z 343.377,A -85,B 0,C 180,E1 -5963.878,E2 -5963.878} C_VEL
LIN {X 0,Y 624.895,Z 343.382,A -85,B 0,C 180,E1 -5967.028,E2 -5967.028} C_VEL
LIN {X 0,Y 624.957,Z 343.384,A -85,B 0,C 180,E1 -5970.053,E2 -5970.053} C_VEL
LIN {X 0,Y 624.894,Z 343.387,A -85,B 0,C 180,E1 -5973.191,E2 -5973.191} C_VEL
LIN {X 0,Y 624.955,Z 343.384,A -85,B 0,C 180,E1 -5976.257,E2 -5976.257} C_VEL
LIN {X 0,Y 624.895,Z 343.388,A -85,B 0,C 180,E1 -5979.319,E2 -5979.319} C_VEL
LIN {X 0,Y 624.956,Z 343.382,A -85,B 0,C 180,E1 -5982.344,E2 -5982.344} C_VEL
LIN {X 0,Y 624.894,Z 343.386,A -85,B 0,C 180,E1 -5985.402,E2 -5985.402} C_VEL
LIN {X 0,Y 624.961,Z 343.536,A -85,B 0,C 180,E1 -5988.228,E2 -5988.228} C_VEL
LIN {X 0,Y 627.576,Z 350.244,A -85,B 0,C 180,E1 -5989.061,E2 -5989.061} C_VEL
LIN {X 0,Y 640.604,Z 371.149,A -85,B 0,C 180,E1 -5990.371,E2 -5990.371} C_VEL
LIN {X 0,Y 642.415,Z 375.848,A -85,B 0,C 180,E1 -5990.573,E2 -5990.573} C_VEL
LIN {X 0,Y 643.44,Z 383.31,A -85,B 0,C 180,E1 -5990.754,E2 -5990.754} C_VEL
LIN {X 0,Y 643.051,Z 394.722,A -85,B 0,C 180,E1 -5990.887,E2 -5990.887} C_VEL
LIN {X 0,Y 642.355,Z 406.342,A -85,B 0,C 180,E1 -5991.001,E2 -5991.001} C_VEL
LIN {X 0,Y 638.289,Z 656.06,A -85,B 0,C 180,E1 -5994.185,E2 -5994.185} C_VEL
LIN {X 0,Y 636.876,Z 739.477,A -85,B 0,C 180,E1 -5995.258,E2 -5995.258} C_VEL
LIN {X 0,Y 635.923,Z 764.625,A -85,B 0,C 180,E1 -5995.74,E2 -5995.74} C_VEL
LIN {X 0,Y 634.923,Z 784.542,A -85,B 0,C 180,E1 -5996.249,E2 -5996.249} C_VEL
LIN {X 0,Y 633.638,Z 806.999,A -85,B 0,C 180,E1 -5996.962,E2 -5996.962} C_VEL
LIN {X 0,Y 632.018,Z 829.116,A -85,B 0,C 180,E1 -5997.835,E2 -5997.835} C_VEL
LIN {X 0,Y 630.445,Z 850.042,A -85,B 0,C 180,E1 -5998.813,E2 -5998.813} C_VEL
LIN {X 0,Y 628.573,Z 872.078,A -85,B 0,C 180,E1 -6000.034,E2 -6000.034} C_VEL
LIN {X 0,Y 626.991,Z 889.692,A -85,B 0,C 180,E1 -6001.157,E2 -6001.157} C_VEL
LIN {X 0,Y 625.065,Z 910.432,A -85,B 0,C 180,E1 -6002.671,E2 -6002.671} C_VEL
LIN {X 0,Y 623.46,Z 927.671,A -85,B 0,C 180,E1 -6004.122,E2 -6004.122} C_VEL
LIN {X 0,Y 621.779,Z 946.335,A -85,B 0,C 180,E1 -6005.892,E2 -6005.892} C_VEL
LIN {X 0,Y 620.403,Z 962.396,A -85,B 0,C 180,E1 -6007.644,E2 -6007.644} C_VEL
LIN {X 0,Y 619.142,Z 978.092,A -85,B 0,C 180,E1 -6009.584,E2 -6009.584} C_VEL
LIN {X 0,Y 618.161,Z 991.588,A -85,B 0,C 180,E1 -6011.516,E2 -6011.516} C_VEL
LIN {X 0,Y 617.356,Z 1004.497,A -85,B 0,C 180,E1 -6013.631,E2 -6013.631} C_VEL
LIN {X 0,Y 616.791,Z 1014.887,A -85,B 0,C 180,E1 -6015.639,E2 -6015.639} C_VEL
LIN {X 0,Y 616.383,Z 1024.598,A -85,B 0,C 180,E1 -6017.826,E2 -6017.826} C_VEL
LIN {X 0,Y 616.114,Z 1032.368,A -85,B 0,C 180,E1 -6020,E2 -6020} C_VEL
LIN {X 0,Y 615.997,Z 1038.132,A -85,B 0,C 180,E1 -6021.976,E2 -6021.976} C_VEL
LIN {X 0,Y 615.926,Z 1043.317,A -85,B 0,C 180,E1 -6024.352,E2 -6024.352} C_VEL
LIN {X 0,Y 615.914,Z 1046.181,A -85,B 0,C 180,E1 -6026.277,E2 -6026.277} C_VEL
LIN {X 0,Y 615.896,Z 1048.13,A -85,B 0,C 180,E1 -6028.512,E2 -6028.512} C_VEL
LIN {X 0,Y 615.895,Z 1048.361,A -85,B 0,C 180,E1 -6030.651,E2 -6030.651} C_VEL
LIN {X 0,Y 615.901,Z 1047.393,A -85,B 0,C 180,E1 -6032.605,E2 -6032.605} C_VEL
LIN {X 0,Y 615.922,Z 1044.688,A -85,B 0,C 180,E1 -6034.936,E2 -6034.936} C_VEL
LIN {X 0,Y 615.966,Z 1040.788,A -85,B 0,C 180,E1 -6036.993,E2 -6036.993} C_VEL
LIN {X 0,Y 616.056,Z 1035.323,A -85,B 0,C 180,E1 -6039.152,E2 -6039.152} C_VEL
LIN {X 0,Y 616.247,Z 1028.123,A -85,B 0,C 180,E1 -6041.322,E2 -6041.322} C_VEL
LIN {X 0,Y 616.536,Z 1020.534,A -85,B 0,C 180,E1 -6043.219,E2 -6043.219} C_VEL
LIN {X 0,Y 617.06,Z 1009.61,A -85,B 0,C 180,E1 -6045.508,E2 -6045.508} C_VEL
LIN {X 0,Y 617.697,Z 998.802,A -85,B 0,C 180,E1 -6047.426,E2 -6047.426} C_VEL
LIN {X 0,Y 618.627,Z 984.965,A -85,B 0,C 180,E1 -6049.557,E2 -6049.557} C_VEL
LIN {X 0,Y 619.686,Z 971.046,A -85,B 0,C 180,E1 -6051.406,E2 -6051.406} C_VEL
LIN {X 0,Y 621.001,Z 955.493,A -85,B 0,C 180,E1 -6053.234,E2 -6053.234} C_VEL
LIN {X 0,Y 622.431,Z 938.948,A -85,B 0,C 180,E1 -6054.923,E2 -6054.923} C_VEL
LIN {X 0,Y 624.206,Z 919.932,A -85,B 0,C 180,E1 -6056.649,E2 -6056.649} C_VEL
LIN {X 0,Y 625.929,Z 901.238,A -85,B 0,C 180,E1 -6058.115,E2 -6058.115} C_VEL
LIN {X 0,Y 627.753,Z 881.474,A -85,B 0,C 180,E1 -6059.484,E2 -6059.484} C_VEL
LIN {X 0,Y 629.539,Z 860.754,A -85,B 0,C 180,E1 -6060.706,E2 -6060.706} C_VEL
LIN {X 0,Y 631.184,Z 840.733,A -85,B 0,C 180,E1 -6061.731,E2 -6061.731} C_VEL
LIN {X 0,Y 632.86,Z 818.101,A -85,B 0,C 180,E1 -6062.707,E2 -6062.707} C_VEL
LIN {X 0,Y 634.159,Z 797.682,A -85,B 0,C 180,E1 -6063.44,E2 -6063.44} C_VEL
LIN {X 0,Y 635.475,Z 774.025,A -85,B 0,C 180,E1 -6064.131,E2 -6064.131} C_VEL
LIN {X 0,Y 636.473,Z 750.788,A -85,B 0,C 180,E1 -6064.636,E2 -6064.636} C_VEL
LIN {X 0,Y 637.207,Z 726.132,A -85,B 0,C 180,E1 -6065.024,E2 -6065.024} C_VEL
LIN {X 0,Y 641.277,Z 471.699,A -85,B 0,C 180,E1 -6068.247,E2 -6068.247} C_VEL
LIN {X 0,Y 642.514,Z 388.128,A -85,B 0,C 180,E1 -6069.336,E2 -6069.336} C_VEL
LIN {X 0,Y 627.827,Z 363.859,A -85,B 0,C 180,E1 -6070.809,E2 -6070.809} C_VEL
LIN {X 0,Y 619.034,Z 350.028,A -85,B 0,C 180,E1 -6071.734,E2 -6071.734} C_VEL
LIN {X 0,Y 616.95,Z 344.371,A -85,B 0,C 180,E1 -6072.488,E2 -6072.488} C_VEL
LIN {X 0,Y 617.014,Z 344.364,A -85,B 0,C 180,E1 -6075.567,E2 -6075.567} C_VEL
LIN {X 0,Y 616.943,Z 344.342,A -85,B 0,C 180,E1 -6078.624,E2 -6078.624} C_VEL
LIN {X 0,Y 617.019,Z 344.372,A -85,B 0,C 180,E1 -6081.659,E2 -6081.659} C_VEL
LIN {X 0,Y 616.949,Z 344.379,A -85,B 0,C 180,E1 -6084.762,E2 -6084.762} C_VEL
LIN {X 0,Y 617.017,Z 344.37,A -85,B 0,C 180,E1 -6087.781,E2 -6087.781} C_VEL
LIN {X 0,Y 616.949,Z 344.378,A -85,B 0,C 180,E1 -6090.802,E2 -6090.802} C_VEL
LIN {X 0,Y 617.019,Z 344.374,A -85,B 0,C 180,E1 -6093.866,E2 -6093.866} C_VEL
LIN {X 0,Y 616.948,Z 344.369,A -85,B 0,C 180,E1 -6096.908,E2 -6096.908} C_VEL
LIN {X 0,Y 617.015,Z 344.362,A -85,B 0,C 180,E1 -6099.906,E2 -6099.906} C_VEL
LIN {X 0,Y 616.948,Z 344.376,A -85,B 0,C 180,E1 -6102.983,E2 -6102.983} C_VEL
LIN {X 0,Y 617.021,Z 344.371,A -85,B 0,C 180,E1 -6106.027,E2 -6106.027} C_VEL
LIN {X 0,Y 616.948,Z 344.363,A -85,B 0,C 180,E1 -6109.069,E2 -6109.069} C_VEL
LIN {X 0,Y 617.015,Z 344.371,A -85,B 0,C 180,E1 -6112.083,E2 -6112.083} C_VEL
LIN {X 0,Y 616.947,Z 344.373,A -85,B 0,C 180,E1 -6115.166,E2 -6115.166} C_VEL
LIN {X 0,Y 617.013,Z 344.36,A -85,B 0,C 180,E1 -6118.236,E2 -6118.236} C_VEL
LIN {X 0,Y 616.948,Z 344.376,A -85,B 0,C 180,E1 -6121.207,E2 -6121.207} C_VEL
LIN {X 0,Y 617.001,Z 344.366,A -85,B 0,C 180,E1 -6124.182,E2 -6124.182} C_VEL
LIN {X 0,Y 616.947,Z 344.367,A -85,B 0,C 180,E1 -6127.31,E2 -6127.31} C_VEL
LIN {X 0,Y 617.002,Z 344.378,A -85,B 0,C 180,E1 -6130.269,E2 -6130.269} C_VEL
LIN {X 0,Y 616.948,Z 344.372,A -85,B 0,C 180,E1 -6133.401,E2 -6133.401} C_VEL
LIN {X 0,Y 616.992,Z 344.365,A -85,B 0,C 180,E1 -6136.282,E2 -6136.282} C_VEL
LIN {X 0,Y 616.952,Z 344.373,A -85,B 0,C 180,E1 -6139.405,E2 -6139.405} C_VEL
LIN {X 0,Y 616.981,Z 344.374,A -85,B 0,C 180,E1 -6142.286,E2 -6142.286} C_VEL
LIN {X 0,Y 616.954,Z 344.374,A -85,B 0,C 180,E1 -6145.482,E2 -6145.482} C_VEL
LIN {X 0,Y 616.975,Z 344.368,A -85,B 0,C 180,E1 -6148.357,E2 -6148.357} C_VEL
LIN {X 0,Y 616.956,Z 344.37,A -85,B 0,C 180,E1 -6151.518,E2 -6151.518} C_VEL
LIN {X 0,Y 616.965,Z 344.372,A -85,B 0,C 180,E1 -6154.332,E2 -6154.332} C_VEL
LIN {X 0,Y 616.96,Z 344.376,A -85,B 0,C 180,E1 -6157.579,E2 -6157.579} C_VEL
LIN {X 0,Y 616.96,Z 344.348,A -85,B 0,C 180,E1 -6160.411,E2 -6160.411} C_VEL
LIN {X 0,Y 616.96,Z 344.374,A -85,B 0,C 180,E1 -6163.712,E2 -6163.712} C_VEL
LIN {X 0,Y 617.018,Z 344.568,A -85,B 0,C 180,E1 -6165.4,E2 -6165.4} C_VEL
LIN {X 0,Y 625.565,Z 366.019,A -85,B 0,C 180,E1 -6168.078,E2 -6168.078} C_VEL
LIN {X 0,Y 629.087,Z 375.223,A -85,B 0,C 180,E1 -6169.128,E2 -6169.128} C_VEL
LIN {X 0,Y 638.398,Z 391.34,A -85,B 0,C 180,E1 -6170.074,E2 -6170.074} C_VEL
LIN {X 0,Y 642.584,Z 410.063,A -85,B 0,C 180,E1 -6170.649,E2 -6170.649} C_VEL
LIN {X 0,Y 638.254,Z 677.156,A -85,B 0,C 180,E1 -6174.05,E2 -6174.05} C_VEL
LIN {X 0,Y 636.744,Z 767.194,A -85,B 0,C 180,E1 -6175.202,E2 -6175.202} C_VEL
LIN {X 0,Y 635.77,Z 792.544,A -85,B 0,C 180,E1 -6175.683,E2 -6175.683} C_VEL
LIN {X 0,Y 634.742,Z 812.649,A -85,B 0,C 180,E1 -6176.192,E2 -6176.192} C_VEL
LIN {X 0,Y 633.393,Z 836.062,A -85,B 0,C 180,E1 -6176.932,E2 -6176.932} C_VEL
LIN {X 0,Y 631.747,Z 858.718,A -85,B 0,C 180,E1 -6177.825,E2 -6177.825} C_VEL
LIN {X 0,Y 630.134,Z 880.671,A -85,B 0,C 180,E1 -6178.849,E2 -6178.849} C_VEL
LIN {X 0,Y 628.362,Z 901.829,A -85,B 0,C 180,E1 -6180.023,E2 -6180.023} C_VEL
LIN {X 0,Y 626.759,Z 920.378,A -85,B 0,C 180,E1 -6181.198,E2 -6181.198} C_VEL
LIN {X 0,Y 624.84,Z 941.825,A -85,B 0,C 180,E1 -6182.763,E2 -6182.763} C_VEL
LIN {X 0,Y 623.347,Z 958.818,A -85,B 0,C 180,E1 -6184.183,E2 -6184.183} C_VEL
LIN {X 0,Y 621.655,Z 977.671,A -85,B 0,C 180,E1 -6185.988,E2 -6185.988} C_VEL
LIN {X 0,Y 620.366,Z 992.776,A -85,B 0,C 180,E1 -6187.643,E2 -6187.643} C_VEL
LIN {X 0,Y 619.114,Z 1008.411,A -85,B 0,C 180,E1 -6189.583,E2 -6189.583} C_VEL
LIN {X 0,Y 618.144,Z 1021.876,A -85,B 0,C 180,E1 -6191.516,E2 -6191.516} C_VEL
LIN {X 0,Y 617.345,Z 1034.733,A -85,B 0,C 180,E1 -6193.631,E2 -6193.631} C_VEL
LIN {X 0,Y 616.778,Z 1045.099,A -85,B 0,C 180,E1 -6195.639,E2 -6195.639} C_VEL
LIN {X 0,Y 616.385,Z 1054.394,A -85,B 0,C 180,E1 -6197.731,E2 -6197.731} C_VEL
LIN {X 0,Y 616.119,Z 1062.21,A -85,B 0,C 180,E1 -6199.905,E2 -6199.905} C_VEL
LIN {X 0,Y 616.003,Z 1067.999,A -85,B 0,C 180,E1 -6201.882,E2 -6201.882} C_VEL
LIN {X 0,Y 615.936,Z 1073.175,A -85,B 0,C 180,E1 -6204.223,E2 -6204.223} C_VEL
LIN {X 0,Y 615.907,Z 1076.123,A -85,B 0,C 180,E1 -6206.183,E2 -6206.183} C_VEL
LIN {X 0,Y 615.897,Z 1077.969,A -85,B 0,C 180,E1 -6208.232,E2 -6208.232} C_VEL
LIN {X 0,Y 615.893,Z 1078.395,A -85,B 0,C 180,E1 -6210.465,E2 -6210.465} C_VEL
LIN {X 0,Y 615.909,Z 1077.496,A -85,B 0,C 180,E1 -6212.419,E2 -6212.419} C_VEL
LIN {X 0,Y 615.921,Z 1075.085,A -85,B 0,C 180,E1 -6214.656,E2 -6214.656} C_VEL
LIN {X 0,Y 615.947,Z 1071.102,A -85,B 0,C 180,E1 -6216.806,E2 -6216.806} C_VEL
LIN {X 0,Y 616.023,Z 1066.219,A -85,B 0,C 180,E1 -6218.776,E2 -6218.776} C_VEL
LIN {X 0,Y 616.234,Z 1058.661,A -85,B 0,C 180,E1 -6221.133,E2 -6221.133} C_VEL
LIN {X 0,Y 616.531,Z 1050.749,A -85,B 0,C 180,E1 -6223.123,E2 -6223.123} C_VEL
LIN {X 0,Y 617.024,Z 1040.404,A -85,B 0,C 180,E1 -6225.316,E2 -6225.316} C_VEL
LIN {X 0,Y 617.669,Z 1029.115,A -85,B 0,C 180,E1 -6227.329,E2 -6227.329} C_VEL
LIN {X 0,Y 618.549,Z 1016.119,A -85,B 0,C 180,E1 -6229.353,E2 -6229.353} C_VEL
LIN {X 0,Y 619.65,Z 1001.615,A -85,B 0,C 180,E1 -6231.289,E2 -6231.289} C_VEL
LIN {X 0,Y 620.977,Z 985.782,A -85,B 0,C 180,E1 -6233.158,E2 -6233.158} C_VEL
LIN {X 0,Y 622.442,Z 968.823,A -85,B 0,C 180,E1 -6234.89,E2 -6234.89} C_VEL
LIN {X 0,Y 623.88,Z 952.658,A -85,B 0,C 180,E1 -6236.356,E2 -6236.356} C_VEL
LIN {X 0,Y 625.654,Z 932.82,A -85,B 0,C 180,E1 -6237.921,E2 -6237.921} C_VEL
LIN {X 0,Y 627.208,Z 915.192,A -85,B 0,C 180,E1 -6239.145,E2 -6239.145} C_VEL
LIN {X 0,Y 629.064,Z 893.416,A -85,B 0,C 180,E1 -6240.467,E2 -6240.467} C_VEL
LIN {X 0,Y 630.661,Z 873.466,A -85,B 0,C 180,E1 -6241.501,E2 -6241.501} C_VEL
LIN {X 0,Y 632.319,Z 851.797,A -85,B 0,C 180,E1 -6242.47,E2 -6242.47} C_VEL
LIN {X 0,Y 633.816,Z 828.423,A -85,B 0,C 180,E1 -6243.325,E2 -6243.325} C_VEL
LIN {X 0,Y 635.037,Z 807.056,A -85,B 0,C 180,E1 -6243.965,E2 -6243.965} C_VEL
LIN {X 0,Y 636.223,Z 781.505,A -85,B 0,C 180,E1 -6244.548,E2 -6244.548} C_VEL
LIN {X 0,Y 636.948,Z 759.379,A -85,B 0,C 180,E1 -6244.91,E2 -6244.91} C_VEL
LIN {X 0,Y 640.776,Z 516.755,A -85,B 0,C 180,E1 -6247.985,E2 -6247.985} C_VEL
LIN {X 0,Y 642.441,Z 408.65,A -85,B 0,C 180,E1 -6249.381,E2 -6249.381} C_VEL
LIN {X 0,Y 637.987,Z 390.387,A -85,B 0,C 180,E1 -6249.969,E2 -6249.969} C_VEL
LIN {X 0,Y 628.727,Z 374.367,A -85,B 0,C 180,E1 -6250.938,E2 -6250.938} C_VEL
LIN {X 0,Y 621.079,Z 354.698,A -85,B 0,C 180,E1 -6253.307,E2 -6253.307} C_VEL
LIN {X 0,Y 617.006,Z 344.476,A -85,B 0,C 180,E1 -6254.606,E2 -6254.606} C_VEL
LIN {X 0,Y 616.951,Z 344.374,A -85,B 0,C 180,E1 -6257.787,E2 -6257.787} C_VEL
LIN {X 0,Y 616.987,Z 344.367,A -85,B 0,C 180,E1 -6260.679,E2 -6260.679} C_VEL
LIN {X 0,Y 616.949,Z 344.335,A -85,B 0,C 180,E1 -6263.847,E2 -6263.847} C_VEL
LIN {X 0,Y 616.989,Z 344.367,A -85,B 0,C 180,E1 -6266.786,E2 -6266.786} C_VEL
LIN {X 0,Y 616.955,Z 344.376,A -85,B 0,C 180,E1 -6269.947,E2 -6269.947} C_VEL
LIN {X 0,Y 616.98,Z 344.362,A -85,B 0,C 180,E1 -6272.805,E2 -6272.805} C_VEL
LIN {X 0,Y 616.958,Z 344.369,A -85,B 0,C 180,E1 -6275.997,E2 -6275.997} C_VEL
LIN {X 0,Y 616.971,Z 344.374,A -85,B 0,C 180,E1 -6278.813,E2 -6278.813} C_VEL
LIN {X 0,Y 616.961,Z 344.377,A -85,B 0,C 180,E1 -6282.066,E2 -6282.066} C_VEL
LIN {X 0,Y 616.978,Z 344.367,A -85,B 0,C 180,E1 -6284.992,E2 -6284.992} C_VEL
LIN {X 0,Y 616.956,Z 344.366,A -85,B 0,C 180,E1 -6288.217,E2 -6288.217} C_VEL
LIN {X 0,Y 616.984,Z 344.374,A -85,B 0,C 180,E1 -6291.144,E2 -6291.144} C_VEL
LIN {X 0,Y 616.959,Z 344.378,A -85,B 0,C 180,E1 -6294.326,E2 -6294.326} C_VEL
LIN {X 0,Y 616.989,Z 344.362,A -85,B 0,C 180,E1 -6297.306,E2 -6297.306} C_VEL
LIN {X 0,Y 616.957,Z 344.374,A -85,B 0,C 180,E1 -6300.464,E2 -6300.464} C_VEL
LIN {X 0,Y 616.994,Z 344.367,A -85,B 0,C 180,E1 -6303.438,E2 -6303.438} C_VEL
LIN {X 0,Y 616.954,Z 344.363,A -85,B 0,C 180,E1 -6306.608,E2 -6306.608} C_VEL
LIN {X 0,Y 616.992,Z 344.373,A -85,B 0,C 180,E1 -6309.515,E2 -6309.515} C_VEL
LIN {X 0,Y 616.957,Z 344.377,A -85,B 0,C 180,E1 -6312.733,E2 -6312.733} C_VEL
LIN {X 0,Y 616.99,Z 344.365,A -85,B 0,C 180,E1 -6315.606,E2 -6315.606} C_VEL
LIN {X 0,Y 616.962,Z 344.373,A -85,B 0,C 180,E1 -6318.717,E2 -6318.717} C_VEL
LIN {X 0,Y 616.989,Z 344.371,A -85,B 0,C 180,E1 -6321.685,E2 -6321.685} C_VEL
LIN {X 0,Y 616.963,Z 344.375,A -85,B 0,C 180,E1 -6324.828,E2 -6324.828} C_VEL
LIN {X 0,Y 616.986,Z 344.366,A -85,B 0,C 180,E1 -6327.767,E2 -6327.767} C_VEL
LIN {X 0,Y 616.96,Z 344.367,A -85,B 0,C 180,E1 -6330.981,E2 -6330.981} C_VEL
LIN {X 0,Y 617.002,Z 344.371,A -85,B 0,C 180,E1 -6333.993,E2 -6333.993} C_VEL
LIN {X 0,Y 616.96,Z 344.369,A -85,B 0,C 180,E1 -6337.12,E2 -6337.12} C_VEL
LIN {X 0,Y 617.003,Z 344.369,A -85,B 0,C 180,E1 -6340.102,E2 -6340.102} C_VEL
LIN {X 0,Y 616.959,Z 344.376,A -85,B 0,C 180,E1 -6343.279,E2 -6343.279} C_VEL
LIN {X 0,Y 617.015,Z 344.377,A -85,B 0,C 180,E1 -6346.343,E2 -6346.343} C_VEL
LIN {X 0,Y 616.993,Z 344.627,A -85,B 0,C 180,E1 -6347.646,E2 -6347.646} C_VEL
LIN {X 0,Y 619.316,Z 350.497,A -85,B 0,C 180,E1 -6348.393,E2 -6348.393} C_VEL
LIN {X 0,Y 633.186,Z 372.46,A -85,B 0,C 180,E1 -6349.828,E2 -6349.828} C_VEL
LIN {X 0,Y 642.656,Z 388.601,A -85,B 0,C 180,E1 -6350.772,E2 -6350.772} C_VEL
LIN {X 0,Y 642.355,Z 406.342,A -85,B 0,C 180,E1 -6351.001,E2 -6351.001} C_VEL
LIN {X 0,Y 641.463,Z 414.043,A -85,B 0,C 180,E1 -6351.045,E2 -6351.045} C_VEL
LIN {X 0,Y 636.22,Z 434.62,A -85,B 0,C 180,E1 -6350.954,E2 -6350.954} C_VEL
LIN {X 0,Y 635.55,Z 441.225,A -85,B 0,C 180,E1 -6350.999,E2 -6350.999} C_VEL
LIN {X 0,Y 631.205,Z 693.394,A -85,B 0,C 180,E1 -6354.232,E2 -6354.232} C_VEL
LIN {X 0,Y 630.26,Z 742.617,A -85,B 0,C 180,E1 -6354.887,E2 -6354.887} C_VEL
LIN {X 0,Y 629.232,Z 766.425,A -85,B 0,C 180,E1 -6355.366,E2 -6355.366} C_VEL
LIN {X 0,Y 628.17,Z 786.392,A -85,B 0,C 180,E1 -6355.888,E2 -6355.888} C_VEL
LIN {X 0,Y 626.69,Z 809.806,A -85,B 0,C 180,E1 -6356.657,E2 -6356.657} C_VEL
LIN {X 0,Y 625.102,Z 830.472,A -85,B 0,C 180,E1 -6357.49,E2 -6357.49} C_VEL
LIN {X 0,Y 623.374,Z 852.267,A -85,B 0,C 180,E1 -6358.527,E2 -6358.527} C_VEL
LIN {X 0,Y 621.458,Z 873.111,A -85,B 0,C 180,E1 -6359.708,E2 -6359.708} C_VEL
LIN {X 0,Y 619.719,Z 891.377,A -85,B 0,C 180,E1 -6360.892,E2 -6360.892} C_VEL
LIN {X 0,Y 617.613,Z 912.468,A -85,B 0,C 180,E1 -6362.47,E2 -6362.47} C_VEL
LIN {X 0,Y 615.966,Z 929.157,A -85,B 0,C 180,E1 -6363.902,E2 -6363.902} C_VEL
LIN {X 0,Y 614.075,Z 948.256,A -85,B 0,C 180,E1 -6365.775,E2 -6365.775} C_VEL
LIN {X 0,Y 612.557,Z 964.935,A -85,B 0,C 180,E1 -6367.646,E2 -6367.646} C_VEL
LIN {X 0,Y 611.233,Z 980.219,A -85,B 0,C 180,E1 -6369.611,E2 -6369.611} C_VEL
LIN {X 0,Y 610.264,Z 992.86,A -85,B 0,C 180,E1 -6371.467,E2 -6371.467} C_VEL
LIN {X 0,Y 609.376,Z 1006.122,A -85,B 0,C 180,E1 -6373.719,E2 -6373.719} C_VEL
LIN {X 0,Y 608.813,Z 1016.064,A -85,B 0,C 180,E1 -6375.696,E2 -6375.696} C_VEL
LIN {X 0,Y 608.369,Z 1026.023,A -85,B 0,C 180,E1 -6378.048,E2 -6378.048} C_VEL
LIN {X 0,Y 608.118,Z 1032.976,A -85,B 0,C 180,E1 -6380.058,E2 -6380.058} C_VEL
LIN {X 0,Y 607.979,Z 1039.141,A -85,B 0,C 180,E1 -6382.25,E2 -6382.25} C_VEL
LIN {X 0,Y 607.924,Z 1043.578,A -85,B 0,C 180,E1 -6384.431,E2 -6384.431} C_VEL
LIN {X 0,Y 607.913,Z 1046.409,A -85,B 0,C 180,E1 -6386.417,E2 -6386.417} C_VEL
LIN {X 0,Y 607.906,Z 1048.202,A -85,B 0,C 180,E1 -6388.775,E2 -6388.775} C_VEL
LIN {X 0,Y 607.899,Z 1048.337,A -85,B 0,C 180,E1 -6390.754,E2 -6390.754} C_VEL
LIN {X 0,Y 607.899,Z 1047.324,A -85,B 0,C 180,E1 -6392.734,E2 -6392.734} C_VEL
LIN {X 0,Y 607.924,Z 1044.528,A -85,B 0,C 180,E1 -6395.096,E2 -6395.096} C_VEL
LIN {X 0,Y 607.976,Z 1040.787,A -85,B 0,C 180,E1 -6397.085,E2 -6397.085} C_VEL
LIN {X 0,Y 608.077,Z 1035.322,A -85,B 0,C 180,E1 -6399.273,E2 -6399.273} C_VEL
LIN {X 0,Y 608.285,Z 1028.121,A -85,B 0,C 180,E1 -6401.473,E2 -6401.473} C_VEL
LIN {X 0,Y 608.6,Z 1020.349,A -85,B 0,C 180,E1 -6403.438,E2 -6403.438} C_VEL
LIN {X 0,Y 609.189,Z 1009.09,A -85,B 0,C 180,E1 -6405.811,E2 -6405.811} C_VEL
LIN {X 0,Y 609.891,Z 998.223,A -85,B 0,C 180,E1 -6407.755,E2 -6407.755} C_VEL
LIN {X 0,Y 610.971,Z 983.628,A -85,B 0,C 180,E1 -6410.001,E2 -6410.001} C_VEL
LIN {X 0,Y 612.051,Z 970.415,A -85,B 0,C 180,E1 -6411.768,E2 -6411.768} C_VEL
LIN {X 0,Y 613.572,Z 953.643,A -85,B 0,C 180,E1 -6413.736,E2 -6413.736} C_VEL
LIN {X 0,Y 615.049,Z 938.298,A -85,B 0,C 180,E1 -6415.325,E2 -6415.325} C_VEL
LIN {X 0,Y 616.927,Z 919.789,A -85,B 0,C 180,E1 -6417.019,E2 -6417.019} C_VEL
LIN {X 0,Y 618.723,Z 901.448,A -85,B 0,C 180,E1 -6418.473,E2 -6418.473} C_VEL
LIN {X 0,Y 620.666,Z 881.682,A -85,B 0,C 180,E1 -6419.854,E2 -6419.854} C_VEL
LIN {X 0,Y 622.569,Z 860.959,A -85,B 0,C 180,E1 -6421.088,E2 -6421.088} C_VEL
LIN {X 0,Y 624.307,Z 840.937,A -85,B 0,C 180,E1 -6422.123,E2 -6422.123} C_VEL
LIN {X 0,Y 626.079,Z 818.301,A -85,B 0,C 180,E1 -6423.107,E2 -6423.107} C_VEL
LIN {X 0,Y 627.459,Z 797.731,A -85,B 0,C 180,E1 -6423.851,E2 -6423.851} C_VEL
LIN {X 0,Y 628.871,Z 773.668,A -85,B 0,C 180,E1 -6424.554,E2 -6424.554} C_VEL
LIN {X 0,Y 629.898,Z 750.97,A -85,B 0,C 180,E1 -6425.05,E2 -6425.05} C_VEL
LIN {X 0,Y 630.666,Z 726.362,A -85,B 0,C 180,E1 -6425.44,E2 -6425.44} C_VEL
LIN {X 0,Y 635.01,Z 471.748,A -85,B 0,C 180,E1 -6428.696,E2 -6428.696} C_VEL
LIN {X 0,Y 636.304,Z 391.294,A -85,B 0,C 180,E1 -6429.753,E2 -6429.753} C_VEL
LIN {X 0,Y 622.466,Z 368.498,A -85,B 0,C 180,E1 -6431.169,E2 -6431.169} C_VEL
LIN {X 0,Y 611.973,Z 352.292,A -85,B 0,C 180,E1 -6432.29,E2 -6432.29} C_VEL
LIN {X 0,Y 610.675,Z 349.99,A -85,B 0,C 180,E1 -6432.47,E2 -6432.47} C_VEL
LIN {X 0,Y 609.038,Z 345.338,A -85,B 0,C 180,E1 -6433.108,E2 -6433.108} C_VEL
LIN {X 0,Y 609.022,Z 345.371,A -85,B 0,C 180,E1 -6436.275,E2 -6436.275} C_VEL
LIN {X 0,Y 609.038,Z 345.328,A -85,B 0,C 180,E1 -6439.2,E2 -6439.2} C_VEL
LIN {X 0,Y 609.02,Z 345.36,A -85,B 0,C 180,E1 -6442.356,E2 -6442.356} C_VEL
LIN {X 0,Y 609.037,Z 345.361,A -85,B 0,C 180,E1 -6445.271,E2 -6445.271} C_VEL
LIN {X 0,Y 609.017,Z 345.359,A -85,B 0,C 180,E1 -6448.527,E2 -6448.527} C_VEL
LIN {X 0,Y 609.045,Z 345.364,A -85,B 0,C 180,E1 -6451.441,E2 -6451.441} C_VEL
LIN {X 0,Y 609.016,Z 345.365,A -85,B 0,C 180,E1 -6454.627,E2 -6454.627} C_VEL
LIN {X 0,Y 609.047,Z 345.36,A -85,B 0,C 180,E1 -6457.562,E2 -6457.562} C_VEL
LIN {X 0,Y 609.016,Z 345.356,A -85,B 0,C 180,E1 -6460.742,E2 -6460.742} C_VEL
LIN {X 0,Y 609.048,Z 345.359,A -85,B 0,C 180,E1 -6463.696,E2 -6463.696} C_VEL
LIN {X 0,Y 609.017,Z 345.365,A -85,B 0,C 180,E1 -6466.808,E2 -6466.808} C_VEL
LIN {X 0,Y 609.045,Z 345.352,A -85,B 0,C 180,E1 -6469.787,E2 -6469.787} C_VEL
LIN {X 0,Y 609.014,Z 345.357,A -85,B 0,C 180,E1 -6472.927,E2 -6472.927} C_VEL
LIN {X 0,Y 609.044,Z 345.365,A -85,B 0,C 180,E1 -6475.858,E2 -6475.858} C_VEL
LIN {X 0,Y 609.014,Z 345.356,A -85,B 0,C 180,E1 -6479.07,E2 -6479.07} C_VEL
LIN {X 0,Y 609.044,Z 345.361,A -85,B 0,C 180,E1 -6481.976,E2 -6481.976} C_VEL
LIN {X 0,Y 609.014,Z 345.365,A -85,B 0,C 180,E1 -6485.181,E2 -6485.181} C_VEL
LIN {X 0,Y 609.049,Z 345.352,A -85,B 0,C 180,E1 -6488.126,E2 -6488.126} C_VEL
LIN {X 0,Y 609.014,Z 345.36,A -85,B 0,C 180,E1 -6491.267,E2 -6491.267} C_VEL
LIN {X 0,Y 609.054,Z 345.365,A -85,B 0,C 180,E1 -6494.256,E2 -6494.256} C_VEL
LIN {X 0,Y 609.012,Z 345.358,A -85,B 0,C 180,E1 -6497.386,E2 -6497.386} C_VEL
LIN {X 0,Y 609.054,Z 345.353,A -85,B 0,C 180,E1 -6500.368,E2 -6500.368} C_VEL
LIN {X 0,Y 609.017,Z 345.361,A -85,B 0,C 180,E1 -6503.411,E2 -6503.411} C_VEL
LIN {X 0,Y 609.039,Z 345.366,A -85,B 0,C 180,E1 -6506.313,E2 -6506.313} C_VEL
LIN {X 0,Y 609.018,Z 345.366,A -85,B 0,C 180,E1 -6509.523,E2 -6509.523} C_VEL
LIN {X 0,Y 609.04,Z 345.364,A -85,B 0,C 180,E1 -6512.45,E2 -6512.45} C_VEL
LIN {X 0,Y 609.015,Z 345.368,A -85,B 0,C 180,E1 -6515.651,E2 -6515.651} C_VEL
LIN {X 0,Y 609.047,Z 345.368,A -85,B 0,C 180,E1 -6518.605,E2 -6518.605} C_VEL
LIN {X 0,Y 609.009,Z 345.344,A -85,B 0,C 180,E1 -6521.807,E2 -6521.807} C_VEL
LIN {X 0,Y 609.067,Z 345.475,A -85,B 0,C 180,E1 -6524.772,E2 -6524.772} C_VEL
LIN {X 0,Y 617.455,Z 366.428,A -85,B 0,C 180,E1 -6527.461,E2 -6527.461} C_VEL
LIN {X 0,Y 620.816,Z 374.906,A -85,B 0,C 180,E1 -6528.463,E2 -6528.463} C_VEL
LIN {X 0,Y 632.714,Z 395.344,A -85,B 0,C 180,E1 -6529.703,E2 -6529.703} C_VEL
LIN {X 0,Y 636.348,Z 411.985,A -85,B 0,C 180,E1 -6530.218,E2 -6530.218} C_VEL
LIN {X 0,Y 631.747,Z 678.218,A -85,B 0,C 180,E1 -6533.638,E2 -6533.638} C_VEL
LIN {X 0,Y 630.156,Z 767.114,A -85,B 0,C 180,E1 -6534.786,E2 -6534.786} C_VEL
LIN {X 0,Y 629.121,Z 792.432,A -85,B 0,C 180,E1 -6535.271,E2 -6535.271} C_VEL
LIN {X 0,Y 628.02,Z 812.759,A -85,B 0,C 180,E1 -6535.79,E2 -6535.79} C_VEL
LIN {X 0,Y 626.576,Z 836.208,A -85,B 0,C 180,E1 -6536.54,E2 -6536.54} C_VEL
LIN {X 0,Y 624.878,Z 858.387,A -85,B 0,C 180,E1 -6537.422,E2 -6537.422} C_VEL
LIN {X 0,Y 623.134,Z 880.452,A -85,B 0,C 180,E1 -6538.459,E2 -6538.459} C_VEL
LIN {X 0,Y 621.253,Z 901.61,A -85,B 0,C 180,E1 -6539.644,E2 -6539.644} C_VEL
LIN {X 0,Y 619.549,Z 920.158,A -85,B 0,C 180,E1 -6540.83,E2 -6540.83} C_VEL
LIN {X 0,Y 617.49,Z 941.604,A -85,B 0,C 180,E1 -6542.412,E2 -6542.412} C_VEL
LIN {X 0,Y 615.94,Z 958.037,A -85,B 0,C 180,E1 -6543.797,E2 -6543.797} C_VEL
LIN {X 0,Y 614.203,Z 976.677,A -85,B 0,C 180,E1 -6545.575,E2 -6545.575} C_VEL
LIN {X 0,Y 612.845,Z 991.46,A -85,B 0,C 180,E1 -6547.196,E2 -6547.196} C_VEL
LIN {X 0,Y 611.522,Z 1006.996,A -85,B 0,C 180,E1 -6549.118,E2 -6549.118} C_VEL
LIN {X 0,Y 610.387,Z 1021.239,A -85,B 0,C 180,E1 -6551.173,E2 -6551.173} C_VEL
LIN {X 0,Y 609.531,Z 1033.688,A -85,B 0,C 180,E1 -6553.219,E2 -6553.219} C_VEL
LIN {X 0,Y 608.879,Z 1044.639,A -85,B 0,C 180,E1 -6555.351,E2 -6555.351} C_VEL
LIN {X 0,Y 608.463,Z 1053.583,A -85,B 0,C 180,E1 -6557.375,E2 -6557.375} C_VEL
LIN {X 0,Y 608.158,Z 1061.907,A -85,B 0,C 180,E1 -6559.676,E2 -6559.676} C_VEL
LIN {X 0,Y 608.023,Z 1067.49,A -85,B 0,C 180,E1 -6561.584,E2 -6561.584} C_VEL
LIN {X 0,Y 607.945,Z 1072.696,A -85,B 0,C 180,E1 -6563.863,E2 -6563.863} C_VEL
LIN {X 0,Y 607.909,Z 1076.009,A -85,B 0,C 180,E1 -6566.039,E2 -6566.039} C_VEL
LIN {X 0,Y 607.906,Z 1077.836,A -85,B 0,C 180,E1 -6568.02,E2 -6568.02} C_VEL
LIN {X 0,Y 607.895,Z 1078.417,A -85,B 0,C 180,E1 -6570.377,E2 -6570.377} C_VEL
LIN {X 0,Y 607.908,Z 1077.495,A -85,B 0,C 180,E1 -6572.451,E2 -6572.451} C_VEL
LIN {X 0,Y 607.923,Z 1075.085,A -85,B 0,C 180,E1 -6574.717,E2 -6574.717} C_VEL
LIN {X 0,Y 607.957,Z 1071.102,A -85,B 0,C 180,E1 -6576.896,E2 -6576.896} C_VEL
LIN {X 0,Y 608.034,Z 1066.219,A -85,B 0,C 180,E1 -6578.892,E2 -6578.892} C_VEL
LIN {X 0,Y 608.266,Z 1058.66,A -85,B 0,C 180,E1 -6581.281,E2 -6581.281} C_VEL
LIN {X 0,Y 608.587,Z 1050.749,A -85,B 0,C 180,E1 -6583.298,E2 -6583.298} C_VEL
LIN {X 0,Y 609.123,Z 1040.403,A -85,B 0,C 180,E1 -6585.52,E2 -6585.52} C_VEL
LIN {X 0,Y 609.827,Z 1029.113,A -85,B 0,C 180,E1 -6587.559,E2 -6587.559} C_VEL
LIN {X 0,Y 610.779,Z 1016.117,A -85,B 0,C 180,E1 -6589.609,E2 -6589.609} C_VEL
LIN {X 0,Y 611.957,Z 1001.613,A -85,B 0,C 180,E1 -6591.57,E2 -6591.57} C_VEL
LIN {X 0,Y 613.373,Z 986,A -85,B 0,C 180,E1 -6593.438,E2 -6593.438} C_VEL
LIN {X 0,Y 614.906,Z 968.972,A -85,B 0,C 180,E1 -6595.186,E2 -6595.186} C_VEL
LIN {X 0,Y 616.66,Z 950.758,A -85,B 0,C 180,E1 -6596.845,E2 -6596.845} C_VEL
LIN {X 0,Y 618.487,Z 931.254,A -85,B 0,C 180,E1 -6598.379,E2 -6598.379} C_VEL
LIN {X 0,Y 620.297,Z 912.011,A -85,B 0,C 180,E1 -6599.714,E2 -6599.714} C_VEL
LIN {X 0,Y 622.246,Z 890.481,A -85,B 0,C 180,E1 -6600.998,E2 -6600.998} C_VEL
LIN {X 0,Y 623.869,Z 871.367,A -85,B 0,C 180,E1 -6601.985,E2 -6601.985} C_VEL
